gfCNCPoint4[28789] = {X 133.2007, Y 6.4835, Z -6.3333, A 0.000, B 0.000, C 0.000 }
gfCNCPoint4[28790] = {X 133.8833, Y 6.4837, Z -6.3333, A 0.000, B 0.000, C 0.000 }
gfCNCPoint4[28791] = {X 134.6792, Y 6.5720, Z -6.3333, A 0.000, B 0.000, C 0.000 }
gfCNCPoint4[28792] = {X 135.4415, Y 6.8171, Z -6.3333, A 0.000, B 0.000, C 0.000 }
gfCNCPoint4[28793] = {X 136.1397, Y 7.2091, Z -6.3333, A 0.000, B 0.000, C 0.000 }
gfCNCPoint4[28794] = {X 136.7458, Y 7.7322, Z -6.3333, A 0.000, B 0.000, C 0.000 }
gfCNCPoint4[28795] = {X 137.2357, Y 8.3657, Z -6.3333, A 0.000, B 0.000, C 0.000 }
gfCNCPoint4[28796] = {X 155.2276, Y 8.3657, Z -6.3333, A 0.000, B 0.000, C 0.000 }
gfCNCPoint4[28797] = {X 155.2814, Y 8.3748, Z -6.3333, A 0.000, B 0.000, C 0.000 }
gfCNCPoint4[28798] = {X 155.3395, Y 8.2839, Z -6.3333, A 0.000, B 0.000, C 0.000 }
gfCNCPoint4[28799] = {X 155.4001, Y 8.1946, Z -6.3333, A 0.000, B 0.000, C 0.000 }
gfCNCPoint4[28800] = {X 156.0394, Y 7.4794, Z -6.3333, A 0.000, B 0.000, C 0.000 }
gfCNCPoint4[28801] = {X 156.8306, Y 6.9370, Z -6.3333, A 0.000, B 0.000, C 0.000 }
gfCNCPoint4[28802] = {X 157.7282, Y 6.5985, Z -6.3333, A 0.000, B 0.000, C 0.000 }
gfCNCPoint4[28803] = {X 158.6805, Y 6.4835, Z -6.3333, A 0.000, B 0.000, C 0.000 }
gfCNCPoint4[28804] = {X 159.3739, Y 6.4839, Z -6.3333, A 0.000, B 0.000, C 0.000 }
gfCNCPoint4[28805] = {X 160.2554, Y 6.5939, Z -6.3333, A 0.000, B 0.000, C 0.000 }
gfCNCPoint4[28806] = {X 161.0909, Y 6.8959, Z -6.3333, A 0.000, B 0.000, C 0.000 }
gfCNCPoint4[28807] = {X 161.8391, Y 7.3747, Z -6.3333, A 0.000, B 0.000, C 0.000 }
gfCNCPoint4[28808] = {X 162.4632, Y 8.0070, Z -6.3333, A 0.000, B 0.000, C 0.000 }
gfCNCPoint4[28809] = {X 162.9324, Y 8.7613, Z -6.3333, A 0.000, B 0.000, C 0.000 }
gfCNCPoint4[28810] = {X 163.2234, Y 9.6007, Z -6.3333, A 0.000, B 0.000, C 0.000 }
gfCNCPoint4[28811] = {X 163.3221, Y 10.4835, Z -6.3333, A 0.000, B 0.000, C 0.000 }
gfCNCPoint4[28812] = {X 163.3221, Y 17.4615, Z -6.3333, A 0.000, B 0.000, C 0.000 }
gfCNCPoint4[28813] = {X 163.2218, Y 18.3516, Z -6.3333, A 0.000, B 0.000, C 0.000 }
gfCNCPoint4[28814] = {X 162.9260, Y 19.1971, Z -6.3333, A 0.000, B 0.000, C 0.000 }
gfCNCPoint4[28815] = {X 162.4494, Y 19.9555, Z -6.3333, A 0.000, B 0.000, C 0.000 }
gfCNCPoint4[28816] = {X 161.8160, Y 20.5889, Z -6.3333, A 0.000, B 0.000, C 0.000 }
gfCNCPoint4[28817] = {X 161.0576, Y 21.0654, Z -6.3333, A 0.000, B 0.000, C 0.000 }
gfCNCPoint4[28818] = {X 160.2122, Y 21.3613, Z -6.3333, A 0.000, B 0.000, C 0.000 }
gfCNCPoint4[28819] = {X 159.3221, Y 21.4615, Z -6.3333, A 0.000, B 0.000, C 0.000 }
gfCNCPoint4[28820] = {X 158.6805, Y 21.4615, Z -6.3333, A 0.000, B 0.000, C 0.000 }
gfCNCPoint4[28821] = {X 157.8710, Y 21.3764, Z -6.3333, A 0.000, B 0.000, C 0.000 }
gfCNCPoint4[28822] = {X 157.0951, Y 21.1304, Z -6.3333, A 0.000, B 0.000, C 0.000 }
gfCNCPoint4[28823] = {X 156.3845, Y 20.7335, Z -6.3333, A 0.000, B 0.000, C 0.000 }
gfCNCPoint4[28824] = {X 155.7680, Y 20.2020, Z -6.3333, A 0.000, B 0.000, C 0.000 }
gfCNCPoint4[28825] = {X 155.2709, Y 19.5575, Z -6.3333, A 0.000, B 0.000, C 0.000 }
gfCNCPoint4[28826] = {X 151.9570, Y 19.5587, Z -6.3333, A 0.000, B 0.000, C 0.000 }
gfCNCPoint4[28827] = {X 151.9558, Y 40.9999, Z -6.3333, A 0.000, B 0.000, C 0.000 }
gfCNCPoint4[28828] = {X 152.5009, Y 41.5868, Z -6.3333, A 0.000, B 0.000, C 0.000 }
gfCNCPoint4[28829] = {X 152.5894, Y 41.6922, Z -6.3333, A 0.000, B 0.000, C 0.000 }
gfCNCPoint4[28830] = {X 153.0754, Y 42.4562, Z -6.3333, A 0.000, B 0.000, C 0.000 }
gfCNCPoint4[28831] = {X 153.3784, Y 43.3095, Z -6.3333, A 0.000, B 0.000, C 0.000 }
gfCNCPoint4[28832] = {X 153.4831, Y 44.2089, Z -6.3333, A 0.000, B 0.000, C 0.000 }
gfCNCPoint4[28833] = {X 153.4829, Y 45.0384, Z -6.3333, A 0.000, B 0.000, C 0.000 }
gfCNCPoint4[28834] = {X 153.3753, Y 45.9222, Z -6.3333, A 0.000, B 0.000, C 0.000 }
gfCNCPoint4[28835] = {X 153.0750, Y 46.7602, Z -6.3333, A 0.000, B 0.000, C 0.000 }
gfCNCPoint4[28836] = {X 152.5967, Y 47.5111, Z -6.3333, A 0.000, B 0.000, C 0.000 }
gfCNCPoint4[28837] = {X 151.9642, Y 48.1376, Z -6.3333, A 0.000, B 0.000, C 0.000 }
gfCNCPoint4[28838] = {X 151.2087, Y 48.6086, Z -6.3333, A 0.000, B 0.000, C 0.000 }
gfCNCPoint4[28839] = {X 150.3678, Y 48.9009, Z -6.3333, A 0.000, B 0.000, C 0.000 }
gfCNCPoint4[28840] = {X 149.4831, Y 49.0000, Z -6.3333, A 0.000, B 0.000, C 0.000 }
gfCNCPoint4[28841] = {X 143.0396, Y 49.0000, Z -6.3333, A 0.000, B 0.000, C 0.000 }
gfCNCPoint4[28842] = {X 142.1495, Y 48.8997, Z -6.3333, A 0.000, B 0.000, C 0.000 }
gfCNCPoint4[28843] = {X 141.3041, Y 48.6039, Z -6.3333, A 0.000, B 0.000, C 0.000 }
gfCNCPoint4[28844] = {X 140.5457, Y 48.1273, Z -6.3333, A 0.000, B 0.000, C 0.000 }
gfCNCPoint4[28845] = {X 139.9123, Y 47.4939, Z -6.3333, A 0.000, B 0.000, C 0.000 }
gfCNCPoint4[28846] = {X 139.4357, Y 46.7355, Z -6.3333, A 0.000, B 0.000, C 0.000 }
gfCNCPoint4[28847] = {X 139.1399, Y 45.8901, Z -6.3333, A 0.000, B 0.000, C 0.000 }
gfCNCPoint4[28848] = {X 139.0396, Y 45.0000, Z -6.3333, A 0.000, B 0.000, C 0.000 }
gfCNCPoint4[28849] = {X 139.0400, Y 44.1538, Z -6.3333, A 0.000, B 0.000, C 0.000 }
gfCNCPoint4[28850] = {X 139.1506, Y 43.2730, Z -6.3333, A 0.000, B 0.000, C 0.000 }
gfCNCPoint4[28851] = {X 139.4528, Y 42.4382, Z -6.3333, A 0.000, B 0.000, C 0.000 }
gfCNCPoint4[28852] = {X 139.9317, Y 41.6907, Z -6.3333, A 0.000, B 0.000, C 0.000 }
gfCNCPoint4[28853] = {X 140.5636, Y 41.0672, Z -6.3333, A 0.000, B 0.000, C 0.000 }
gfCNCPoint4[28854] = {X 140.5636, Y 30.3968, Z -6.3333, A 0.000, B 0.000, C 0.000 }
gfCNCPoint4[28855] = {X 136.4836, Y 30.3968, Z -6.3333, A 0.000, B 0.000, C 0.000 }
gfCNCPoint4[28856] = {X 136.4836, Y 30.3968, Z -3.3333, A 0.000, B 0.000, C 0.000 }
gfCNCPoint4[28857] = {X 136.4836, Y 30.3968, Z 11.0000, A 0.000, B 0.000, C 0.000 }
gfCNCPoint4[28858] = {X 137.6634, Y 74.8921, Z 11.0000, A 0.000, B 0.000, C 0.000 }
gfCNCPoint4[28859] = {X 137.6634, Y 74.8921, Z -3.3333, A 0.000, B 0.000, C 0.000 }
gfCNCPoint4[28860] = {X 137.6634, Y 74.8921, Z -6.3333, A 0.000, B 0.000, C 0.000 }
gfCNCPoint4[28861] = {X 140.6800, Y 77.6392, Z -6.3333, A 0.000, B 0.000, C 0.000 }
gfCNCPoint4[28862] = {X 155.6321, Y 61.2197, Z -6.3333, A 0.000, B 0.000, C 0.000 }
gfCNCPoint4[28863] = {X 155.2773, Y 60.5141, Z -6.3333, A 0.000, B 0.000, C 0.000 }
gfCNCPoint4[28864] = {X 155.0568, Y 59.7556, Z -6.3333, A 0.000, B 0.000, C 0.000 }
gfCNCPoint4[28865] = {X 154.9781, Y 58.9697, Z -6.3333, A 0.000, B 0.000, C 0.000 }
gfCNCPoint4[28866] = {X 154.9780, Y 58.0000, Z -6.3333, A 0.000, B 0.000, C 0.000 }
gfCNCPoint4[28867] = {X 155.0863, Y 57.0387, Z -6.3333, A 0.000, B 0.000, C 0.000 }
gfCNCPoint4[28868] = {X 155.4058, Y 56.1256, Z -6.3333, A 0.000, B 0.000, C 0.000 }
gfCNCPoint4[28869] = {X 155.9204, Y 55.3065, Z -6.3333, A 0.000, B 0.000, C 0.000 }
gfCNCPoint4[28870] = {X 156.6045, Y 54.6225, Z -6.3333, A 0.000, B 0.000, C 0.000 }
gfCNCPoint4[28871] = {X 157.4236, Y 54.1078, Z -6.3333, A 0.000, B 0.000, C 0.000 }
gfCNCPoint4[28872] = {X 158.3367, Y 53.7883, Z -6.3333, A 0.000, B 0.000, C 0.000 }
gfCNCPoint4[28873] = {X 159.2980, Y 53.6800, Z -6.3333, A 0.000, B 0.000, C 0.000 }
gfCNCPoint4[28874] = {X 178.5335, Y 53.6800, Z -6.3333, A 0.000, B 0.000, C 0.000 }
gfCNCPoint4[28875] = {X 179.4948, Y 53.7883, Z -6.3333, A 0.000, B 0.000, C 0.000 }
gfCNCPoint4[28876] = {X 180.4079, Y 54.1078, Z -6.3333, A 0.000, B 0.000, C 0.000 }
gfCNCPoint4[28877] = {X 181.2270, Y 54.6225, Z -6.3333, A 0.000, B 0.000, C 0.000 }
gfCNCPoint4[28878] = {X 181.9110, Y 55.3065, Z -6.3333, A 0.000, B 0.000, C 0.000 }
gfCNCPoint4[28879] = {X 182.4257, Y 56.1256, Z -6.3333, A 0.000, B 0.000, C 0.000 }
gfCNCPoint4[28880] = {X 182.7452, Y 57.0387, Z -6.3333, A 0.000, B 0.000, C 0.000 }
gfCNCPoint4[28881] = {X 182.8535, Y 58.0000, Z -6.3333, A 0.000, B 0.000, C 0.000 }
gfCNCPoint4[28882] = {X 182.8535, Y 58.9342, Z -6.3333, A 0.000, B 0.000, C 0.000 }
gfCNCPoint4[28883] = {X 182.7808, Y 59.7231, Z -6.3333, A 0.000, B 0.000, C 0.000 }
gfCNCPoint4[28884] = {X 182.5653, Y 60.4855, Z -6.3333, A 0.000, B 0.000, C 0.000 }
gfCNCPoint4[28885] = {X 182.2142, Y 61.1956, Z -6.3333, A 0.000, B 0.000, C 0.000 }
gfCNCPoint4[28886] = {X 209.4796, Y 90.9543, Z -6.3333, A 0.000, B 0.000, C 0.000 }
gfCNCPoint4[28887] = {X 210.1361, Y 91.6204, Z -6.3333, A 0.000, B 0.000, C 0.000 }
gfCNCPoint4[28888] = {X 210.8392, Y 92.2369, Z -6.3333, A 0.000, B 0.000, C 0.000 }
gfCNCPoint4[28889] = {X 211.1136, Y 92.4105, Z -6.3333, A 0.000, B 0.000, C 0.000 }
gfCNCPoint4[28890] = {X 211.4212, Y 92.5146, Z -6.3333, A 0.000, B 0.000, C 0.000 }
gfCNCPoint4[28891] = {X 213.4040, Y 92.8239, Z -6.3333, A 0.000, B 0.000, C 0.000 }
gfCNCPoint4[28892] = {X 214.4546, Y 92.7351, Z -6.3333, A 0.000, B 0.000, C 0.000 }
gfCNCPoint4[28893] = {X 215.5073, Y 92.6749, Z -6.3333, A 0.000, B 0.000, C 0.000 }
gfCNCPoint4[28894] = {X 216.1774, Y 92.6018, Z -6.3333, A 0.000, B 0.000, C 0.000 }
gfCNCPoint4[28895] = {X 216.8226, Y 92.4068, Z -6.3333, A 0.000, B 0.000, C 0.000 }
gfCNCPoint4[28896] = {X 217.4209, Y 92.0964, Z -6.3333, A 0.000, B 0.000, C 0.000 }
gfCNCPoint4[28897] = {X 222.9613, Y 88.5209, Z -6.3333, A 0.000, B 0.000, C 0.000 }
gfCNCPoint4[28898] = {X 245.8274, Y 73.8996, Z -6.3333, A 0.000, B 0.000, C 0.000 }
gfCNCPoint4[28899] = {X 221.6306, Y 64.4044, Z -6.3333, A 0.000, B 0.000, C 0.000 }
gfCNCPoint4[28900] = {X 219.8631, Y 63.8129, Z -6.3333, A 0.000, B 0.000, C 0.000 }
gfCNCPoint4[28901] = {X 218.0397, Y 63.4269, Z -6.3333, A 0.000, B 0.000, C 0.000 }
gfCNCPoint4[28902] = {X 216.1841, Y 63.2516, Z -6.3333, A 0.000, B 0.000, C 0.000 }
gfCNCPoint4[28903] = {X 215.2523, Y 63.1173, Z -6.3333, A 0.000, B 0.000, C 0.000 }
gfCNCPoint4[28904] = {X 214.3716, Y 62.7843, Z -6.3333, A 0.000, B 0.000, C 0.000 }
gfCNCPoint4[28905] = {X 213.5841, Y 62.2684, Z -6.3333, A 0.000, B 0.000, C 0.000 }
gfCNCPoint4[28906] = {X 212.9270, Y 61.5942, Z -6.3333, A 0.000, B 0.000, C 0.000 }
gfCNCPoint4[28907] = {X 212.4315, Y 60.7936, Z -6.3333, A 0.000, B 0.000, C 0.000 }
gfCNCPoint4[28908] = {X 212.1213, Y 59.9047, Z -6.3333, A 0.000, B 0.000, C 0.000 }
gfCNCPoint4[28909] = {X 212.0110, Y 58.9697, Z -6.3333, A 0.000, B 0.000, C 0.000 }
gfCNCPoint4[28910] = {X 212.0108, Y 58.0000, Z -6.3333, A 0.000, B 0.000, C 0.000 }
gfCNCPoint4[28911] = {X 212.1191, Y 57.0387, Z -6.3333, A 0.000, B 0.000, C 0.000 }
gfCNCPoint4[28912] = {X 212.4386, Y 56.1256, Z -6.3333, A 0.000, B 0.000, C 0.000 }
gfCNCPoint4[28913] = {X 212.9533, Y 55.3065, Z -6.3333, A 0.000, B 0.000, C 0.000 }
gfCNCPoint4[28914] = {X 213.6373, Y 54.6225, Z -6.3333, A 0.000, B 0.000, C 0.000 }
gfCNCPoint4[28915] = {X 214.4564, Y 54.1078, Z -6.3333, A 0.000, B 0.000, C 0.000 }
gfCNCPoint4[28916] = {X 215.3695, Y 53.7883, Z -6.3333, A 0.000, B 0.000, C 0.000 }
gfCNCPoint4[28917] = {X 216.3308, Y 53.6800, Z -6.3333, A 0.000, B 0.000, C 0.000 }
gfCNCPoint4[28918] = {X 237.2617, Y 53.6800, Z -6.3333, A 0.000, B 0.000, C 0.000 }
gfCNCPoint4[28919] = {X 238.2230, Y 53.7883, Z -6.3333, A 0.000, B 0.000, C 0.000 }
gfCNCPoint4[28920] = {X 239.1361, Y 54.1078, Z -6.3333, A 0.000, B 0.000, C 0.000 }
gfCNCPoint4[28921] = {X 239.9552, Y 54.6225, Z -6.3333, A 0.000, B 0.000, C 0.000 }
gfCNCPoint4[28922] = {X 240.6392, Y 55.3065, Z -6.3333, A 0.000, B 0.000, C 0.000 }
gfCNCPoint4[28923] = {X 241.1539, Y 56.1256, Z -6.3333, A 0.000, B 0.000, C 0.000 }
gfCNCPoint4[28924] = {X 241.4734, Y 57.0387, Z -6.3333, A 0.000, B 0.000, C 0.000 }
gfCNCPoint4[28925] = {X 241.5817, Y 58.0000, Z -6.3333, A 0.000, B 0.000, C 0.000 }
gfCNCPoint4[28926] = {X 241.5817, Y 58.2319, Z -6.3333, A 0.000, B 0.000, C 0.000 }
gfCNCPoint4[28927] = {X 248.1145, Y 60.7793, Z -6.3333, A 0.000, B 0.000, C 0.000 }
gfCNCPoint4[28928] = {X 275.6322, Y 71.7016, Z -6.3333, A 0.000, B 0.000, C 0.000 }
gfCNCPoint4[28929] = {X 275.6336, Y 63.2123, Z -6.3333, A 0.000, B 0.000, C 0.000 }
gfCNCPoint4[28930] = {X 274.7820, Y 63.0032, Z -6.3333, A 0.000, B 0.000, C 0.000 }
gfCNCPoint4[28931] = {X 273.9901, Y 62.6264, Z -6.3333, A 0.000, B 0.000, C 0.000 }
gfCNCPoint4[28932] = {X 273.2907, Y 62.0974, Z -6.3333, A 0.000, B 0.000, C 0.000 }
gfCNCPoint4[28933] = {X 272.7125, Y 61.4381, Z -6.3333, A 0.000, B 0.000, C 0.000 }
gfCNCPoint4[28934] = {X 272.2793, Y 60.6756, Z -6.3333, A 0.000, B 0.000, C 0.000 }
gfCNCPoint4[28935] = {X 272.0090, Y 59.8414, Z -6.3333, A 0.000, B 0.000, C 0.000 }
gfCNCPoint4[28936] = {X 271.9128, Y 58.9697, Z -6.3333, A 0.000, B 0.000, C 0.000 }
gfCNCPoint4[28937] = {X 271.9127, Y 58.0000, Z -6.3333, A 0.000, B 0.000, C 0.000 }
gfCNCPoint4[28938] = {X 272.0210, Y 57.0387, Z -6.3333, A 0.000, B 0.000, C 0.000 }
gfCNCPoint4[28939] = {X 272.3405, Y 56.1256, Z -6.3333, A 0.000, B 0.000, C 0.000 }
gfCNCPoint4[28940] = {X 272.8552, Y 55.3065, Z -6.3333, A 0.000, B 0.000, C 0.000 }
gfCNCPoint4[28941] = {X 273.5392, Y 54.6225, Z -6.3333, A 0.000, B 0.000, C 0.000 }
gfCNCPoint4[28942] = {X 274.3583, Y 54.1078, Z -6.3333, A 0.000, B 0.000, C 0.000 }
gfCNCPoint4[28943] = {X 275.2714, Y 53.7883, Z -6.3333, A 0.000, B 0.000, C 0.000 }
gfCNCPoint4[28944] = {X 276.2327, Y 53.6800, Z -6.3333, A 0.000, B 0.000, C 0.000 }
gfCNCPoint4[28945] = {X 292.7731, Y 53.6800, Z -6.3333, A 0.000, B 0.000, C 0.000 }
gfCNCPoint4[28946] = {X 293.7344, Y 53.7883, Z -6.3333, A 0.000, B 0.000, C 0.000 }
gfCNCPoint4[28947] = {X 294.6475, Y 54.1078, Z -6.3333, A 0.000, B 0.000, C 0.000 }
gfCNCPoint4[28948] = {X 295.4666, Y 54.6225, Z -6.3333, A 0.000, B 0.000, C 0.000 }
gfCNCPoint4[28949] = {X 296.1506, Y 55.3065, Z -6.3333, A 0.000, B 0.000, C 0.000 }
gfCNCPoint4[28950] = {X 296.6653, Y 56.1256, Z -6.3333, A 0.000, B 0.000, C 0.000 }
gfCNCPoint4[28951] = {X 296.9848, Y 57.0387, Z -6.3333, A 0.000, B 0.000, C 0.000 }
gfCNCPoint4[28952] = {X 297.0931, Y 58.0000, Z -6.3333, A 0.000, B 0.000, C 0.000 }
gfCNCPoint4[28953] = {X 297.0931, Y 58.9350, Z -6.3333, A 0.000, B 0.000, C 0.000 }
gfCNCPoint4[28954] = {X 296.9713, Y 59.9431, Z -6.3333, A 0.000, B 0.000, C 0.000 }
gfCNCPoint4[28955] = {X 296.6183, Y 60.8953, Z -6.3333, A 0.000, B 0.000, C 0.000 }
gfCNCPoint4[28956] = {X 296.0536, Y 61.7393, Z -6.3333, A 0.000, B 0.000, C 0.000 }
gfCNCPoint4[28957] = {X 295.3082, Y 62.4288, Z -6.3333, A 0.000, B 0.000, C 0.000 }
gfCNCPoint4[28958] = {X 294.4227, Y 62.9260, Z -6.3333, A 0.000, B 0.000, C 0.000 }
gfCNCPoint4[28959] = {X 293.4460, Y 63.2036, Z -6.3333, A 0.000, B 0.000, C 0.000 }
gfCNCPoint4[28960] = {X 293.3735, Y 63.2251, Z -6.3333, A 0.000, B 0.000, C 0.000 }
gfCNCPoint4[28961] = {X 293.3847, Y 92.7805, Z -6.3333, A 0.000, B 0.000, C 0.000 }
gfCNCPoint4[28962] = {X 294.2373, Y 92.9980, Z -6.3333, A 0.000, B 0.000, C 0.000 }
gfCNCPoint4[28963] = {X 295.0288, Y 93.3825, Z -6.3333, A 0.000, B 0.000, C 0.000 }
gfCNCPoint4[28964] = {X 295.7267, Y 93.9184, Z -6.3333, A 0.000, B 0.000, C 0.000 }
gfCNCPoint4[28965] = {X 296.3026, Y 94.5837, Z -6.3333, A 0.000, B 0.000, C 0.000 }
gfCNCPoint4[28966] = {X 296.7329, Y 95.3512, Z -6.3333, A 0.000, B 0.000, C 0.000 }
gfCNCPoint4[28967] = {X 297.0000, Y 96.1896, Z -6.3333, A 0.000, B 0.000, C 0.000 }
gfCNCPoint4[28968] = {X 297.0931, Y 97.0645, Z -6.3333, A 0.000, B 0.000, C 0.000 }
gfCNCPoint4[28969] = {X 297.0931, Y 98.0000, Z -6.3333, A 0.000, B 0.000, C 0.000 }
gfCNCPoint4[28970] = {X 296.9848, Y 98.9613, Z -6.3333, A 0.000, B 0.000, C 0.000 }
gfCNCPoint4[28971] = {X 296.6653, Y 99.8744, Z -6.3333, A 0.000, B 0.000, C 0.000 }
gfCNCPoint4[28972] = {X 296.1506, Y 100.6935, Z -6.3333, A 0.000, B 0.000, C 0.000 }
gfCNCPoint4[28973] = {X 295.4666, Y 101.3775, Z -6.3333, A 0.000, B 0.000, C 0.000 }
gfCNCPoint4[28974] = {X 294.6475, Y 101.8922, Z -6.3333, A 0.000, B 0.000, C 0.000 }
gfCNCPoint4[28975] = {X 293.7344, Y 102.2117, Z -6.3333, A 0.000, B 0.000, C 0.000 }
gfCNCPoint4[28976] = {X 292.7731, Y 102.3200, Z -6.3333, A 0.000, B 0.000, C 0.000 }
gfCNCPoint4[28977] = {X 276.2327, Y 102.3200, Z -6.3333, A 0.000, B 0.000, C 0.000 }
gfCNCPoint4[28978] = {X 275.2714, Y 102.2117, Z -6.3333, A 0.000, B 0.000, C 0.000 }
gfCNCPoint4[28979] = {X 274.3583, Y 101.8922, Z -6.3333, A 0.000, B 0.000, C 0.000 }
gfCNCPoint4[28980] = {X 273.5392, Y 101.3775, Z -6.3333, A 0.000, B 0.000, C 0.000 }
gfCNCPoint4[28981] = {X 272.8552, Y 100.6935, Z -6.3333, A 0.000, B 0.000, C 0.000 }
gfCNCPoint4[28982] = {X 272.3405, Y 99.8744, Z -6.3333, A 0.000, B 0.000, C 0.000 }
gfCNCPoint4[28983] = {X 272.0210, Y 98.9613, Z -6.3333, A 0.000, B 0.000, C 0.000 }
gfCNCPoint4[28984] = {X 271.9127, Y 98.0000, Z -6.3333, A 0.000, B 0.000, C 0.000 }
gfCNCPoint4[28985] = {X 271.9127, Y 97.0659, Z -6.3333, A 0.000, B 0.000, C 0.000 }
gfCNCPoint4[28986] = {X 272.0026, Y 96.1891, Z -6.3333, A 0.000, B 0.000, C 0.000 }
gfCNCPoint4[28987] = {X 272.2686, Y 95.3488, Z -6.3333, A 0.000, B 0.000, C 0.000 }
gfCNCPoint4[28988] = {X 272.6997, Y 94.5800, Z -6.3333, A 0.000, B 0.000, C 0.000 }
gfCNCPoint4[28989] = {X 273.2777, Y 93.9146, Z -6.3333, A 0.000, B 0.000, C 0.000 }
gfCNCPoint4[28990] = {X 273.9788, Y 93.3805, Z -6.3333, A 0.000, B 0.000, C 0.000 }
gfCNCPoint4[28991] = {X 274.7737, Y 92.9997, Z -6.3333, A 0.000, B 0.000, C 0.000 }
gfCNCPoint4[28992] = {X 275.6294, Y 92.7883, Z -6.3333, A 0.000, B 0.000, C 0.000 }
gfCNCPoint4[28993] = {X 275.6294, Y 85.5950, Z -6.3333, A 0.000, B 0.000, C 0.000 }
gfCNCPoint4[28994] = {X 262.6398, Y 80.5030, Z -6.3333, A 0.000, B 0.000, C 0.000 }
gfCNCPoint4[28995] = {X 262.2779, Y 80.7315, Z -6.3333, A 0.000, B 0.000, C 0.000 }
gfCNCPoint4[28996] = {X 237.7972, Y 96.5883, Z -6.3333, A 0.000, B 0.000, C 0.000 }
gfCNCPoint4[28997] = {X 237.7998, Y 97.0650, Z -6.3333, A 0.000, B 0.000, C 0.000 }
gfCNCPoint4[28998] = {X 237.7998, Y 98.0000, Z -6.3333, A 0.000, B 0.000, C 0.000 }
gfCNCPoint4[28999] = {X 237.6915, Y 98.9613, Z -6.3333, A 0.000, B 0.000, C 0.000 }
gfCNCPoint4[29000] = {X 237.3720, Y 99.8744, Z -6.3333, A 0.000, B 0.000, C 0.000 }
gfCNCPoint4[29001] = {X 236.8573, Y 100.6935, Z -6.3333, A 0.000, B 0.000, C 0.000 }
gfCNCPoint4[29002] = {X 236.1733, Y 101.3775, Z -6.3333, A 0.000, B 0.000, C 0.000 }
gfCNCPoint4[29003] = {X 235.3542, Y 101.8922, Z -6.3333, A 0.000, B 0.000, C 0.000 }
gfCNCPoint4[29004] = {X 234.4411, Y 102.2117, Z -6.3333, A 0.000, B 0.000, C 0.000 }
gfCNCPoint4[29005] = {X 233.4798, Y 102.3200, Z -6.3333, A 0.000, B 0.000, C 0.000 }
gfCNCPoint4[29006] = {X 214.1790, Y 102.3200, Z -6.3333, A 0.000, B 0.000, C 0.000 }
gfCNCPoint4[29007] = {X 213.7862, Y 102.3021, Z -6.3333, A 0.000, B 0.000, C 0.000 }
gfCNCPoint4[29008] = {X 213.3966, Y 102.2485, Z -6.3333, A 0.000, B 0.000, C 0.000 }
gfCNCPoint4[29009] = {X 213.0070, Y 102.3021, Z -6.3333, A 0.000, B 0.000, C 0.000 }
gfCNCPoint4[29010] = {X 212.6141, Y 102.3200, Z -6.3333, A 0.000, B 0.000, C 0.000 }
gfCNCPoint4[29011] = {X 194.9870, Y 102.3200, Z -6.3333, A 0.000, B 0.000, C 0.000 }
gfCNCPoint4[29012] = {X 194.0257, Y 102.2117, Z -6.3333, A 0.000, B 0.000, C 0.000 }
gfCNCPoint4[29013] = {X 193.1126, Y 101.8922, Z -6.3333, A 0.000, B 0.000, C 0.000 }
gfCNCPoint4[29014] = {X 192.2935, Y 101.3775, Z -6.3333, A 0.000, B 0.000, C 0.000 }
gfCNCPoint4[29015] = {X 191.6094, Y 100.6935, Z -6.3333, A 0.000, B 0.000, C 0.000 }
gfCNCPoint4[29016] = {X 191.0948, Y 99.8744, Z -6.3333, A 0.000, B 0.000, C 0.000 }
gfCNCPoint4[29017] = {X 190.7753, Y 98.9613, Z -6.3333, A 0.000, B 0.000, C 0.000 }
gfCNCPoint4[29018] = {X 190.6670, Y 98.0000, Z -6.3333, A 0.000, B 0.000, C 0.000 }
gfCNCPoint4[29019] = {X 190.6670, Y 97.0659, Z -6.3333, A 0.000, B 0.000, C 0.000 }
gfCNCPoint4[29020] = {X 190.7727, Y 96.1162, Z -6.3333, A 0.000, B 0.000, C 0.000 }
gfCNCPoint4[29021] = {X 191.0846, Y 95.2129, Z -6.3333, A 0.000, B 0.000, C 0.000 }
gfCNCPoint4[29022] = {X 191.5874, Y 94.4003, Z -6.3333, A 0.000, B 0.000, C 0.000 }
gfCNCPoint4[29023] = {X 188.5647, Y 91.1002, Z -6.3333, A 0.000, B 0.000, C 0.000 }
gfCNCPoint4[29024] = {X 150.0898, Y 91.1002, Z -6.3333, A 0.000, B 0.000, C 0.000 }
gfCNCPoint4[29025] = {X 147.1454, Y 94.3623, Z -6.3333, A 0.000, B 0.000, C 0.000 }
gfCNCPoint4[29026] = {X 147.6646, Y 95.1836, Z -6.3333, A 0.000, B 0.000, C 0.000 }
gfCNCPoint4[29027] = {X 147.9879, Y 96.1000, Z -6.3333, A 0.000, B 0.000, C 0.000 }
gfCNCPoint4[29028] = {X 148.0991, Y 97.0653, Z -6.3333, A 0.000, B 0.000, C 0.000 }
gfCNCPoint4[29029] = {X 148.0991, Y 98.0000, Z -6.3333, A 0.000, B 0.000, C 0.000 }
gfCNCPoint4[29030] = {X 147.9908, Y 98.9613, Z -6.3333, A 0.000, B 0.000, C 0.000 }
gfCNCPoint4[29031] = {X 147.6713, Y 99.8744, Z -6.3333, A 0.000, B 0.000, C 0.000 }
gfCNCPoint4[29032] = {X 147.1566, Y 100.6935, Z -6.3333, A 0.000, B 0.000, C 0.000 }
gfCNCPoint4[29033] = {X 146.4726, Y 101.3775, Z -6.3333, A 0.000, B 0.000, C 0.000 }
gfCNCPoint4[29034] = {X 145.6535, Y 101.8922, Z -6.3333, A 0.000, B 0.000, C 0.000 }
gfCNCPoint4[29035] = {X 144.7404, Y 102.2117, Z -6.3333, A 0.000, B 0.000, C 0.000 }
gfCNCPoint4[29036] = {X 143.7791, Y 102.3200, Z -6.3333, A 0.000, B 0.000, C 0.000 }
gfCNCPoint4[29037] = {X 125.0000, Y 102.3200, Z -6.3333, A 0.000, B 0.000, C 0.000 }
gfCNCPoint4[29038] = {X 124.0387, Y 102.2117, Z -6.3333, A 0.000, B 0.000, C 0.000 }
gfCNCPoint4[29039] = {X 123.1256, Y 101.8922, Z -6.3333, A 0.000, B 0.000, C 0.000 }
gfCNCPoint4[29040] = {X 122.3065, Y 101.3775, Z -6.3333, A 0.000, B 0.000, C 0.000 }
gfCNCPoint4[29041] = {X 121.6225, Y 100.6935, Z -6.3333, A 0.000, B 0.000, C 0.000 }
gfCNCPoint4[29042] = {X 121.1078, Y 99.8744, Z -6.3333, A 0.000, B 0.000, C 0.000 }
gfCNCPoint4[29043] = {X 120.7883, Y 98.9613, Z -6.3333, A 0.000, B 0.000, C 0.000 }
gfCNCPoint4[29044] = {X 120.6800, Y 98.0000, Z -6.3333, A 0.000, B 0.000, C 0.000 }
gfCNCPoint4[29045] = {X 120.6800, Y 97.0659, Z -6.3333, A 0.000, B 0.000, C 0.000 }
gfCNCPoint4[29046] = {X 120.7832, Y 96.1275, Z -6.3333, A 0.000, B 0.000, C 0.000 }
gfCNCPoint4[29047] = {X 121.0877, Y 95.2340, Z -6.3333, A 0.000, B 0.000, C 0.000 }
gfCNCPoint4[29048] = {X 121.5790, Y 94.4279, Z -6.3333, A 0.000, B 0.000, C 0.000 }
gfCNCPoint4[29049] = {X 122.2338, Y 93.7478, Z -6.3333, A 0.000, B 0.000, C 0.000 }
gfCNCPoint4[29050] = {X 123.0206, Y 93.2261, Z -6.3333, A 0.000, B 0.000, C 0.000 }
gfCNCPoint4[29051] = {X 123.9019, Y 92.8878, Z -6.3333, A 0.000, B 0.000, C 0.000 }
gfCNCPoint4[29052] = {X 124.8357, Y 92.7491, Z -6.3333, A 0.000, B 0.000, C 0.000 }
gfCNCPoint4[29053] = {X 124.8807, Y 92.7315, Z -6.3333, A 0.000, B 0.000, C 0.000 }
gfCNCPoint4[29054] = {X 124.9278, Y 92.7208, Z -6.3333, A 0.000, B 0.000, C 0.000 }
gfCNCPoint4[29055] = {X 125.4494, Y 92.6434, Z -6.3333, A 0.000, B 0.000, C 0.000 }
gfCNCPoint4[29056] = {X 126.2804, Y 92.5036, Z -6.3333, A 0.000, B 0.000, C 0.000 }
gfCNCPoint4[29057] = {X 127.0999, Y 92.3072, Z -6.3333, A 0.000, B 0.000, C 0.000 }
gfCNCPoint4[29058] = {X 128.3213, Y 91.1562, Z -6.3333, A 0.000, B 0.000, C 0.000 }
gfCNCPoint4[29059] = {X 129.4782, Y 89.9403, Z -6.3333, A 0.000, B 0.000, C 0.000 }
gfCNCPoint4[29060] = {X 140.6800, Y 77.6392, Z -6.3333, A 0.000, B 0.000, C 0.000 }
gfCNCPoint4[29061] = {X 137.7225, Y 74.9460, Z -6.3333, A 0.000, B 0.000, C 0.000 }
gfCNCPoint4[29062] = {X 140.7391, Y 77.6930, Z -6.3333, A 0.000, B 0.000, C 0.000 }
gfCNCPoint4[29063] = {X 155.7324, Y 61.2284, Z -6.3333, A 0.000, B 0.000, C 0.000 }
gfCNCPoint4[29064] = {X 155.3666, Y 60.5223, Z -6.3333, A 0.000, B 0.000, C 0.000 }
gfCNCPoint4[29065] = {X 155.1392, Y 59.7602, Z -6.3333, A 0.000, B 0.000, C 0.000 }
gfCNCPoint4[29066] = {X 155.0581, Y 58.9691, Z -6.3333, A 0.000, B 0.000, C 0.000 }
gfCNCPoint4[29067] = {X 155.0580, Y 58.0000, Z -6.3333, A 0.000, B 0.000, C 0.000 }
gfCNCPoint4[29068] = {X 155.1643, Y 57.0565, Z -6.3333, A 0.000, B 0.000, C 0.000 }
gfCNCPoint4[29069] = {X 155.4778, Y 56.1603, Z -6.3333, A 0.000, B 0.000, C 0.000 }
gfCNCPoint4[29070] = {X 155.9830, Y 55.3564, Z -6.3333, A 0.000, B 0.000, C 0.000 }
gfCNCPoint4[29071] = {X 156.6544, Y 54.6850, Z -6.3333, A 0.000, B 0.000, C 0.000 }
gfCNCPoint4[29072] = {X 157.4583, Y 54.1799, Z -6.3333, A 0.000, B 0.000, C 0.000 }
gfCNCPoint4[29073] = {X 158.3545, Y 53.8663, Z -6.3333, A 0.000, B 0.000, C 0.000 }
gfCNCPoint4[29074] = {X 159.2980, Y 53.7600, Z -6.3333, A 0.000, B 0.000, C 0.000 }
gfCNCPoint4[29075] = {X 178.5335, Y 53.7600, Z -6.3333, A 0.000, B 0.000, C 0.000 }
gfCNCPoint4[29076] = {X 179.4770, Y 53.8663, Z -6.3333, A 0.000, B 0.000, C 0.000 }
gfCNCPoint4[29077] = {X 180.3732, Y 54.1799, Z -6.3333, A 0.000, B 0.000, C 0.000 }
gfCNCPoint4[29078] = {X 181.1771, Y 54.6850, Z -6.3333, A 0.000, B 0.000, C 0.000 }
gfCNCPoint4[29079] = {X 181.8485, Y 55.3564, Z -6.3333, A 0.000, B 0.000, C 0.000 }
gfCNCPoint4[29080] = {X 182.3536, Y 56.1603, Z -6.3333, A 0.000, B 0.000, C 0.000 }
gfCNCPoint4[29081] = {X 182.6672, Y 57.0565, Z -6.3333, A 0.000, B 0.000, C 0.000 }
gfCNCPoint4[29082] = {X 182.7735, Y 58.0000, Z -6.3333, A 0.000, B 0.000, C 0.000 }
gfCNCPoint4[29083] = {X 182.7735, Y 58.9342, Z -6.3333, A 0.000, B 0.000, C 0.000 }
gfCNCPoint4[29084] = {X 182.6985, Y 59.7282, Z -6.3333, A 0.000, B 0.000, C 0.000 }
gfCNCPoint4[29085] = {X 182.4761, Y 60.4941, Z -6.3333, A 0.000, B 0.000, C 0.000 }
gfCNCPoint4[29086] = {X 182.1142, Y 61.2048, Z -6.3333, A 0.000, B 0.000, C 0.000 }
gfCNCPoint4[29087] = {X 209.4206, Y 91.0084, Z -6.3333, A 0.000, B 0.000, C 0.000 }
gfCNCPoint4[29088] = {X 210.0812, Y 91.6786, Z -6.3333, A 0.000, B 0.000, C 0.000 }
gfCNCPoint4[29089] = {X 210.7887, Y 92.2989, Z -6.3333, A 0.000, B 0.000, C 0.000 }
gfCNCPoint4[29090] = {X 211.0801, Y 92.4832, Z -6.3333, A 0.000, B 0.000, C 0.000 }
gfCNCPoint4[29091] = {X 211.4068, Y 92.5933, Z -6.3333, A 0.000, B 0.000, C 0.000 }
gfCNCPoint4[29092] = {X 213.4017, Y 92.9045, Z -6.3333, A 0.000, B 0.000, C 0.000 }
gfCNCPoint4[29093] = {X 214.4547, Y 92.8153, Z -6.3333, A 0.000, B 0.000, C 0.000 }
gfCNCPoint4[29094] = {X 215.5097, Y 92.7549, Z -6.3333, A 0.000, B 0.000, C 0.000 }
gfCNCPoint4[29095] = {X 216.1941, Y 92.6801, Z -6.3333, A 0.000, B 0.000, C 0.000 }
gfCNCPoint4[29096] = {X 216.8531, Y 92.4807, Z -6.3333, A 0.000, B 0.000, C 0.000 }
gfCNCPoint4[29097] = {X 217.4643, Y 92.1637, Z -6.3333, A 0.000, B 0.000, C 0.000 }
gfCNCPoint4[29098] = {X 223.0046, Y 88.5882, Z -6.3333, A 0.000, B 0.000, C 0.000 }
gfCNCPoint4[29099] = {X 246.0027, Y 73.8825, Z -6.3333, A 0.000, B 0.000, C 0.000 }
gfCNCPoint4[29100] = {X 221.6603, Y 64.3301, Z -6.3333, A 0.000, B 0.000, C 0.000 }
gfCNCPoint4[29101] = {X 219.8841, Y 63.7357, Z -6.3333, A 0.000, B 0.000, C 0.000 }
gfCNCPoint4[29102] = {X 218.0517, Y 63.3478, Z -6.3333, A 0.000, B 0.000, C 0.000 }
gfCNCPoint4[29103] = {X 216.1870, Y 63.1716, Z -6.3333, A 0.000, B 0.000, C 0.000 }
gfCNCPoint4[29104] = {X 215.2724, Y 63.0398, Z -6.3333, A 0.000, B 0.000, C 0.000 }
gfCNCPoint4[29105] = {X 214.4080, Y 62.7130, Z -6.3333, A 0.000, B 0.000, C 0.000 }
gfCNCPoint4[29106] = {X 213.6350, Y 62.2067, Z -6.3333, A 0.000, B 0.000, C 0.000 }
gfCNCPoint4[29107] = {X 212.9900, Y 61.5450, Z -6.3333, A 0.000, B 0.000, C 0.000 }
gfCNCPoint4[29108] = {X 212.5038, Y 60.7592, Z -6.3333, A 0.000, B 0.000, C 0.000 }
gfCNCPoint4[29109] = {X 212.1992, Y 59.8868, Z -6.3333, A 0.000, B 0.000, C 0.000 }
gfCNCPoint4[29110] = {X 212.0910, Y 58.9691, Z -6.3333, A 0.000, B 0.000, C 0.000 }
gfCNCPoint4[29111] = {X 212.0908, Y 58.0000, Z -6.3333, A 0.000, B 0.000, C 0.000 }
gfCNCPoint4[29112] = {X 212.1971, Y 57.0565, Z -6.3333, A 0.000, B 0.000, C 0.000 }
gfCNCPoint4[29113] = {X 212.5107, Y 56.1603, Z -6.3333, A 0.000, B 0.000, C 0.000 }
gfCNCPoint4[29114] = {X 213.0158, Y 55.3564, Z -6.3333, A 0.000, B 0.000, C 0.000 }
gfCNCPoint4[29115] = {X 213.6872, Y 54.6850, Z -6.3333, A 0.000, B 0.000, C 0.000 }
gfCNCPoint4[29116] = {X 214.4911, Y 54.1799, Z -6.3333, A 0.000, B 0.000, C 0.000 }
gfCNCPoint4[29117] = {X 215.3873, Y 53.8663, Z -6.3333, A 0.000, B 0.000, C 0.000 }
gfCNCPoint4[29118] = {X 216.3308, Y 53.7600, Z -6.3333, A 0.000, B 0.000, C 0.000 }
gfCNCPoint4[29119] = {X 237.2617, Y 53.7600, Z -6.3333, A 0.000, B 0.000, C 0.000 }
gfCNCPoint4[29120] = {X 238.2052, Y 53.8663, Z -6.3333, A 0.000, B 0.000, C 0.000 }
gfCNCPoint4[29121] = {X 239.1014, Y 54.1799, Z -6.3333, A 0.000, B 0.000, C 0.000 }
gfCNCPoint4[29122] = {X 239.9053, Y 54.6850, Z -6.3333, A 0.000, B 0.000, C 0.000 }
gfCNCPoint4[29123] = {X 240.5767, Y 55.3564, Z -6.3333, A 0.000, B 0.000, C 0.000 }
gfCNCPoint4[29124] = {X 241.0818, Y 56.1603, Z -6.3333, A 0.000, B 0.000, C 0.000 }
gfCNCPoint4[29125] = {X 241.3954, Y 57.0565, Z -6.3333, A 0.000, B 0.000, C 0.000 }
gfCNCPoint4[29126] = {X 241.5017, Y 58.0000, Z -6.3333, A 0.000, B 0.000, C 0.000 }
gfCNCPoint4[29127] = {X 241.5017, Y 58.2866, Z -6.3333, A 0.000, B 0.000, C 0.000 }
gfCNCPoint4[29128] = {X 248.0852, Y 60.8537, Z -6.3333, A 0.000, B 0.000, C 0.000 }
gfCNCPoint4[29129] = {X 275.7122, Y 71.8194, Z -6.3333, A 0.000, B 0.000, C 0.000 }
gfCNCPoint4[29130] = {X 275.7136, Y 63.1422, Z -6.3333, A 0.000, B 0.000, C 0.000 }
gfCNCPoint4[29131] = {X 274.8651, Y 62.9475, Z -6.3333, A 0.000, B 0.000, C 0.000 }
gfCNCPoint4[29132] = {X 274.0742, Y 62.5835, Z -6.3333, A 0.000, B 0.000, C 0.000 }
gfCNCPoint4[29133] = {X 273.3744, Y 62.0658, Z -6.3333, A 0.000, B 0.000, C 0.000 }
gfCNCPoint4[29134] = {X 272.7950, Y 61.4160, Z -6.3333, A 0.000, B 0.000, C 0.000 }
gfCNCPoint4[29135] = {X 272.3606, Y 60.6616, Z -6.3333, A 0.000, B 0.000, C 0.000 }
gfCNCPoint4[29136] = {X 272.0894, Y 59.8343, Z -6.3333, A 0.000, B 0.000, C 0.000 }
gfCNCPoint4[29137] = {X 271.9928, Y 58.9691, Z -6.3333, A 0.000, B 0.000, C 0.000 }
gfCNCPoint4[29138] = {X 271.9927, Y 58.0000, Z -6.3333, A 0.000, B 0.000, C 0.000 }
gfCNCPoint4[29139] = {X 272.0990, Y 57.0565, Z -6.3333, A 0.000, B 0.000, C 0.000 }
gfCNCPoint4[29140] = {X 272.4126, Y 56.1603, Z -6.3333, A 0.000, B 0.000, C 0.000 }
gfCNCPoint4[29141] = {X 272.9177, Y 55.3564, Z -6.3333, A 0.000, B 0.000, C 0.000 }
gfCNCPoint4[29142] = {X 273.5891, Y 54.6850, Z -6.3333, A 0.000, B 0.000, C 0.000 }
gfCNCPoint4[29143] = {X 274.3930, Y 54.1799, Z -6.3333, A 0.000, B 0.000, C 0.000 }
gfCNCPoint4[29144] = {X 275.2892, Y 53.8663, Z -6.3333, A 0.000, B 0.000, C 0.000 }
gfCNCPoint4[29145] = {X 276.2327, Y 53.7600, Z -6.3333, A 0.000, B 0.000, C 0.000 }
gfCNCPoint4[29146] = {X 292.7731, Y 53.7600, Z -6.3333, A 0.000, B 0.000, C 0.000 }
gfCNCPoint4[29147] = {X 293.7166, Y 53.8663, Z -6.3333, A 0.000, B 0.000, C 0.000 }
gfCNCPoint4[29148] = {X 294.6128, Y 54.1799, Z -6.3333, A 0.000, B 0.000, C 0.000 }
gfCNCPoint4[29149] = {X 295.4167, Y 54.6850, Z -6.3333, A 0.000, B 0.000, C 0.000 }
gfCNCPoint4[29150] = {X 296.0881, Y 55.3564, Z -6.3333, A 0.000, B 0.000, C 0.000 }
gfCNCPoint4[29151] = {X 296.5932, Y 56.1603, Z -6.3333, A 0.000, B 0.000, C 0.000 }
gfCNCPoint4[29152] = {X 296.9068, Y 57.0565, Z -6.3333, A 0.000, B 0.000, C 0.000 }
gfCNCPoint4[29153] = {X 297.0131, Y 58.0000, Z -6.3333, A 0.000, B 0.000, C 0.000 }
gfCNCPoint4[29154] = {X 297.0131, Y 58.9348, Z -6.3333, A 0.000, B 0.000, C 0.000 }
gfCNCPoint4[29155] = {X 296.8933, Y 59.9252, Z -6.3333, A 0.000, B 0.000, C 0.000 }
gfCNCPoint4[29156] = {X 296.5463, Y 60.8604, Z -6.3333, A 0.000, B 0.000, C 0.000 }
gfCNCPoint4[29157] = {X 295.9912, Y 61.6893, Z -6.3333, A 0.000, B 0.000, C 0.000 }
gfCNCPoint4[29158] = {X 295.2583, Y 62.3661, Z -6.3333, A 0.000, B 0.000, C 0.000 }
gfCNCPoint4[29159] = {X 294.3881, Y 62.8538, Z -6.3333, A 0.000, B 0.000, C 0.000 }
gfCNCPoint4[29160] = {X 293.4282, Y 63.1255, Z -6.3333, A 0.000, B 0.000, C 0.000 }
gfCNCPoint4[29161] = {X 293.2934, Y 63.1654, Z -6.3333, A 0.000, B 0.000, C 0.000 }
gfCNCPoint4[29162] = {X 293.3048, Y 92.8500, Z -6.3333, A 0.000, B 0.000, C 0.000 }
gfCNCPoint4[29163] = {X 294.1543, Y 93.0532, Z -6.3333, A 0.000, B 0.000, C 0.000 }
gfCNCPoint4[29164] = {X 294.9447, Y 93.4250, Z -6.3333, A 0.000, B 0.000, C 0.000 }
gfCNCPoint4[29165] = {X 295.6431, Y 93.9498, Z -6.3333, A 0.000, B 0.000, C 0.000 }
gfCNCPoint4[29166] = {X 296.2201, Y 94.6056, Z -6.3333, A 0.000, B 0.000, C 0.000 }
gfCNCPoint4[29167] = {X 296.6516, Y 95.3650, Z -6.3333, A 0.000, B 0.000, C 0.000 }
gfCNCPoint4[29168] = {X 296.9197, Y 96.1964, Z -6.3333, A 0.000, B 0.000, C 0.000 }
gfCNCPoint4[29169] = {X 297.0131, Y 97.0649, Z -6.3333, A 0.000, B 0.000, C 0.000 }
gfCNCPoint4[29170] = {X 297.0131, Y 98.0000, Z -6.3333, A 0.000, B 0.000, C 0.000 }
gfCNCPoint4[29171] = {X 296.9068, Y 98.9435, Z -6.3333, A 0.000, B 0.000, C 0.000 }
gfCNCPoint4[29172] = {X 296.5932, Y 99.8397, Z -6.3333, A 0.000, B 0.000, C 0.000 }
gfCNCPoint4[29173] = {X 296.0881, Y 100.6436, Z -6.3333, A 0.000, B 0.000, C 0.000 }
gfCNCPoint4[29174] = {X 295.4167, Y 101.3150, Z -6.3333, A 0.000, B 0.000, C 0.000 }
gfCNCPoint4[29175] = {X 294.6128, Y 101.8201, Z -6.3333, A 0.000, B 0.000, C 0.000 }
gfCNCPoint4[29176] = {X 293.7166, Y 102.1337, Z -6.3333, A 0.000, B 0.000, C 0.000 }
gfCNCPoint4[29177] = {X 292.7731, Y 102.2400, Z -6.3333, A 0.000, B 0.000, C 0.000 }
gfCNCPoint4[29178] = {X 276.2327, Y 102.2400, Z -6.3333, A 0.000, B 0.000, C 0.000 }
gfCNCPoint4[29179] = {X 275.2892, Y 102.1337, Z -6.3333, A 0.000, B 0.000, C 0.000 }
gfCNCPoint4[29180] = {X 274.3930, Y 101.8201, Z -6.3333, A 0.000, B 0.000, C 0.000 }
gfCNCPoint4[29181] = {X 273.5891, Y 101.3150, Z -6.3333, A 0.000, B 0.000, C 0.000 }
gfCNCPoint4[29182] = {X 272.9177, Y 100.6436, Z -6.3333, A 0.000, B 0.000, C 0.000 }
gfCNCPoint4[29183] = {X 272.4126, Y 99.8397, Z -6.3333, A 0.000, B 0.000, C 0.000 }
gfCNCPoint4[29184] = {X 272.0990, Y 98.9435, Z -6.3333, A 0.000, B 0.000, C 0.000 }
gfCNCPoint4[29185] = {X 271.9927, Y 98.0000, Z -6.3333, A 0.000, B 0.000, C 0.000 }
gfCNCPoint4[29186] = {X 271.9927, Y 97.0659, Z -6.3333, A 0.000, B 0.000, C 0.000 }
gfCNCPoint4[29187] = {X 272.0830, Y 96.1956, Z -6.3333, A 0.000, B 0.000, C 0.000 }
gfCNCPoint4[29188] = {X 272.3500, Y 95.3624, Z -6.3333, A 0.000, B 0.000, C 0.000 }
gfCNCPoint4[29189] = {X 272.7823, Y 94.6017, Z -6.3333, A 0.000, B 0.000, C 0.000 }
gfCNCPoint4[29190] = {X 273.3615, Y 93.9460, Z -6.3333, A 0.000, B 0.000, C 0.000 }
gfCNCPoint4[29191] = {X 274.0630, Y 93.4231, Z -6.3333, A 0.000, B 0.000, C 0.000 }
gfCNCPoint4[29192] = {X 274.8569, Y 93.0553, Z -6.3333, A 0.000, B 0.000, C 0.000 }
gfCNCPoint4[29193] = {X 275.7094, Y 92.8584, Z -6.3333, A 0.000, B 0.000, C 0.000 }
gfCNCPoint4[29194] = {X 275.7094, Y 85.5404, Z -6.3333, A 0.000, B 0.000, C 0.000 }
gfCNCPoint4[29195] = {X 262.6313, Y 80.4138, Z -6.3333, A 0.000, B 0.000, C 0.000 }
gfCNCPoint4[29196] = {X 262.2347, Y 80.6641, Z -6.3333, A 0.000, B 0.000, C 0.000 }
gfCNCPoint4[29197] = {X 237.7169, Y 96.5449, Z -6.3333, A 0.000, B 0.000, C 0.000 }
gfCNCPoint4[29198] = {X 237.7198, Y 97.0652, Z -6.3333, A 0.000, B 0.000, C 0.000 }
gfCNCPoint4[29199] = {X 237.7198, Y 98.0000, Z -6.3333, A 0.000, B 0.000, C 0.000 }
gfCNCPoint4[29200] = {X 237.6135, Y 98.9435, Z -6.3333, A 0.000, B 0.000, C 0.000 }
gfCNCPoint4[29201] = {X 237.2999, Y 99.8397, Z -6.3333, A 0.000, B 0.000, C 0.000 }
gfCNCPoint4[29202] = {X 236.7948, Y 100.6436, Z -6.3333, A 0.000, B 0.000, C 0.000 }
gfCNCPoint4[29203] = {X 236.1234, Y 101.3150, Z -6.3333, A 0.000, B 0.000, C 0.000 }
gfCNCPoint4[29204] = {X 235.3195, Y 101.8201, Z -6.3333, A 0.000, B 0.000, C 0.000 }
gfCNCPoint4[29205] = {X 234.4233, Y 102.1337, Z -6.3333, A 0.000, B 0.000, C 0.000 }
gfCNCPoint4[29206] = {X 233.4798, Y 102.2400, Z -6.3333, A 0.000, B 0.000, C 0.000 }
gfCNCPoint4[29207] = {X 214.1790, Y 102.2400, Z -6.3333, A 0.000, B 0.000, C 0.000 }
gfCNCPoint4[29208] = {X 213.7861, Y 102.2218, Z -6.3333, A 0.000, B 0.000, C 0.000 }
gfCNCPoint4[29209] = {X 213.3966, Y 102.1672, Z -6.3333, A 0.000, B 0.000, C 0.000 }
gfCNCPoint4[29210] = {X 213.0070, Y 102.2218, Z -6.3333, A 0.000, B 0.000, C 0.000 }
gfCNCPoint4[29211] = {X 212.6141, Y 102.2400, Z -6.3333, A 0.000, B 0.000, C 0.000 }
gfCNCPoint4[29212] = {X 194.9870, Y 102.2400, Z -6.3333, A 0.000, B 0.000, C 0.000 }
gfCNCPoint4[29213] = {X 194.0435, Y 102.1337, Z -6.3333, A 0.000, B 0.000, C 0.000 }
gfCNCPoint4[29214] = {X 193.1473, Y 101.8201, Z -6.3333, A 0.000, B 0.000, C 0.000 }
gfCNCPoint4[29215] = {X 192.3434, Y 101.3150, Z -6.3333, A 0.000, B 0.000, C 0.000 }
gfCNCPoint4[29216] = {X 191.6720, Y 100.6436, Z -6.3333, A 0.000, B 0.000, C 0.000 }
gfCNCPoint4[29217] = {X 191.1669, Y 99.8397, Z -6.3333, A 0.000, B 0.000, C 0.000 }
gfCNCPoint4[29218] = {X 190.8533, Y 98.9435, Z -6.3333, A 0.000, B 0.000, C 0.000 }
gfCNCPoint4[29219] = {X 190.7470, Y 98.0000, Z -6.3333, A 0.000, B 0.000, C 0.000 }
gfCNCPoint4[29220] = {X 190.7470, Y 97.0659, Z -6.3333, A 0.000, B 0.000, C 0.000 }
gfCNCPoint4[29221] = {X 190.8557, Y 96.1118, Z -6.3333, A 0.000, B 0.000, C 0.000 }
gfCNCPoint4[29222] = {X 191.1764, Y 95.2065, Z -6.3333, A 0.000, B 0.000, C 0.000 }
gfCNCPoint4[29223] = {X 191.6926, Y 94.3967, Z -6.3333, A 0.000, B 0.000, C 0.000 }
gfCNCPoint4[29224] = {X 188.5999, Y 91.0202, Z -6.3333, A 0.000, B 0.000, C 0.000 }
gfCNCPoint4[29225] = {X 150.0543, Y 91.0202, Z -6.3333, A 0.000, B 0.000, C 0.000 }
gfCNCPoint4[29226] = {X 147.0401, Y 94.3596, Z -6.3333, A 0.000, B 0.000, C 0.000 }
gfCNCPoint4[29227] = {X 147.5726, Y 95.1779, Z -6.3333, A 0.000, B 0.000, C 0.000 }
gfCNCPoint4[29228] = {X 147.9048, Y 96.0959, Z -6.3333, A 0.000, B 0.000, C 0.000 }
gfCNCPoint4[29229] = {X 148.0191, Y 97.0655, Z -6.3333, A 0.000, B 0.000, C 0.000 }
gfCNCPoint4[29230] = {X 148.0191, Y 98.0000, Z -6.3333, A 0.000, B 0.000, C 0.000 }
gfCNCPoint4[29231] = {X 147.9128, Y 98.9435, Z -6.3333, A 0.000, B 0.000, C 0.000 }
gfCNCPoint4[29232] = {X 147.5992, Y 99.8397, Z -6.3333, A 0.000, B 0.000, C 0.000 }
gfCNCPoint4[29233] = {X 147.0941, Y 100.6436, Z -6.3333, A 0.000, B 0.000, C 0.000 }
gfCNCPoint4[29234] = {X 146.4227, Y 101.3150, Z -6.3333, A 0.000, B 0.000, C 0.000 }
gfCNCPoint4[29235] = {X 145.6188, Y 101.8201, Z -6.3333, A 0.000, B 0.000, C 0.000 }
gfCNCPoint4[29236] = {X 144.7226, Y 102.1337, Z -6.3333, A 0.000, B 0.000, C 0.000 }
gfCNCPoint4[29237] = {X 143.7791, Y 102.2400, Z -6.3333, A 0.000, B 0.000, C 0.000 }
gfCNCPoint4[29238] = {X 125.0000, Y 102.2400, Z -6.3333, A 0.000, B 0.000, C 0.000 }
gfCNCPoint4[29239] = {X 124.0565, Y 102.1337, Z -6.3333, A 0.000, B 0.000, C 0.000 }
gfCNCPoint4[29240] = {X 123.1603, Y 101.8201, Z -6.3333, A 0.000, B 0.000, C 0.000 }
gfCNCPoint4[29241] = {X 122.3564, Y 101.3150, Z -6.3333, A 0.000, B 0.000, C 0.000 }
gfCNCPoint4[29242] = {X 121.6850, Y 100.6436, Z -6.3333, A 0.000, B 0.000, C 0.000 }
gfCNCPoint4[29243] = {X 121.1799, Y 99.8397, Z -6.3333, A 0.000, B 0.000, C 0.000 }
gfCNCPoint4[29244] = {X 120.8663, Y 98.9435, Z -6.3333, A 0.000, B 0.000, C 0.000 }
gfCNCPoint4[29245] = {X 120.7600, Y 98.0000, Z -6.3333, A 0.000, B 0.000, C 0.000 }
gfCNCPoint4[29246] = {X 120.7600, Y 97.0659, Z -6.3333, A 0.000, B 0.000, C 0.000 }
gfCNCPoint4[29247] = {X 120.8618, Y 96.1424, Z -6.3333, A 0.000, B 0.000, C 0.000 }
gfCNCPoint4[29248] = {X 121.1623, Y 95.2633, Z -6.3333, A 0.000, B 0.000, C 0.000 }
gfCNCPoint4[29249] = {X 121.6471, Y 94.4707, Z -6.3333, A 0.000, B 0.000, C 0.000 }
gfCNCPoint4[29250] = {X 122.2928, Y 93.8027, Z -6.3333, A 0.000, B 0.000, C 0.000 }
gfCNCPoint4[29251] = {X 123.0686, Y 93.2914, Z -6.3333, A 0.000, B 0.000, C 0.000 }
gfCNCPoint4[29252] = {X 123.9371, Y 92.9613, Z -6.3333, A 0.000, B 0.000, C 0.000 }
gfCNCPoint4[29253] = {X 124.8566, Y 92.8284, Z -6.3333, A 0.000, B 0.000, C 0.000 }
gfCNCPoint4[29254] = {X 124.8968, Y 92.8103, Z -6.3333, A 0.000, B 0.000, C 0.000 }
gfCNCPoint4[29255] = {X 124.9395, Y 92.7999, Z -6.3333, A 0.000, B 0.000, C 0.000 }
gfCNCPoint4[29256] = {X 125.4606, Y 92.7226, Z -6.3333, A 0.000, B 0.000, C 0.000 }
gfCNCPoint4[29257] = {X 126.3058, Y 92.5801, Z -6.3333, A 0.000, B 0.000, C 0.000 }
gfCNCPoint4[29258] = {X 127.1392, Y 92.3793, Z -6.3333, A 0.000, B 0.000, C 0.000 }
gfCNCPoint4[29259] = {X 128.3711, Y 91.2194, Z -6.3333, A 0.000, B 0.000, C 0.000 }
gfCNCPoint4[29260] = {X 129.5377, Y 89.9938, Z -6.3333, A 0.000, B 0.000, C 0.000 }
gfCNCPoint4[29261] = {X 140.7391, Y 77.6930, Z -6.3333, A 0.000, B 0.000, C 0.000 }
gfCNCPoint4[29262] = {X 137.7817, Y 74.9999, Z -6.3333, A 0.000, B 0.000, C 0.000 }
gfCNCPoint4[29263] = {X 140.7983, Y 77.7469, Z -6.3333, A 0.000, B 0.000, C 0.000 }
gfCNCPoint4[29264] = {X 155.8332, Y 61.2365, Z -6.3333, A 0.000, B 0.000, C 0.000 }
gfCNCPoint4[29265] = {X 155.4563, Y 60.5301, Z -6.3333, A 0.000, B 0.000, C 0.000 }
gfCNCPoint4[29266] = {X 155.2217, Y 59.7647, Z -6.3333, A 0.000, B 0.000, C 0.000 }
gfCNCPoint4[29267] = {X 155.1381, Y 58.9684, Z -6.3333, A 0.000, B 0.000, C 0.000 }
gfCNCPoint4[29268] = {X 155.1380, Y 58.0000, Z -6.3333, A 0.000, B 0.000, C 0.000 }
gfCNCPoint4[29269] = {X 155.2423, Y 57.0743, Z -6.3333, A 0.000, B 0.000, C 0.000 }
gfCNCPoint4[29270] = {X 155.5499, Y 56.1950, Z -6.3333, A 0.000, B 0.000, C 0.000 }
gfCNCPoint4[29271] = {X 156.0455, Y 55.4063, Z -6.3333, A 0.000, B 0.000, C 0.000 }
gfCNCPoint4[29272] = {X 156.7042, Y 54.7476, Z -6.3333, A 0.000, B 0.000, C 0.000 }
gfCNCPoint4[29273] = {X 157.4930, Y 54.2520, Z -6.3333, A 0.000, B 0.000, C 0.000 }
gfCNCPoint4[29274] = {X 158.3723, Y 53.9443, Z -6.3333, A 0.000, B 0.000, C 0.000 }
gfCNCPoint4[29275] = {X 159.2980, Y 53.8400, Z -6.3333, A 0.000, B 0.000, C 0.000 }
gfCNCPoint4[29276] = {X 178.5335, Y 53.8400, Z -6.3333, A 0.000, B 0.000, C 0.000 }
gfCNCPoint4[29277] = {X 179.4592, Y 53.9443, Z -6.3333, A 0.000, B 0.000, C 0.000 }
gfCNCPoint4[29278] = {X 180.3385, Y 54.2520, Z -6.3333, A 0.000, B 0.000, C 0.000 }
gfCNCPoint4[29279] = {X 181.1272, Y 54.7476, Z -6.3333, A 0.000, B 0.000, C 0.000 }
gfCNCPoint4[29280] = {X 181.7859, Y 55.4063, Z -6.3333, A 0.000, B 0.000, C 0.000 }
gfCNCPoint4[29281] = {X 182.2815, Y 56.1950, Z -6.3333, A 0.000, B 0.000, C 0.000 }
gfCNCPoint4[29282] = {X 182.5892, Y 57.0743, Z -6.3333, A 0.000, B 0.000, C 0.000 }
gfCNCPoint4[29283] = {X 182.6935, Y 58.0000, Z -6.3333, A 0.000, B 0.000, C 0.000 }
gfCNCPoint4[29284] = {X 182.6935, Y 58.9342, Z -6.3333, A 0.000, B 0.000, C 0.000 }
gfCNCPoint4[29285] = {X 182.6160, Y 59.7333, Z -6.3333, A 0.000, B 0.000, C 0.000 }
gfCNCPoint4[29286] = {X 182.3865, Y 60.5025, Z -6.3333, A 0.000, B 0.000, C 0.000 }
gfCNCPoint4[29287] = {X 182.0135, Y 61.2134, Z -6.3333, A 0.000, B 0.000, C 0.000 }
gfCNCPoint4[29288] = {X 209.3617, Y 91.0624, Z -6.3333, A 0.000, B 0.000, C 0.000 }
gfCNCPoint4[29289] = {X 210.0263, Y 91.7368, Z -6.3333, A 0.000, B 0.000, C 0.000 }
gfCNCPoint4[29290] = {X 210.7382, Y 92.3609, Z -6.3333, A 0.000, B 0.000, C 0.000 }
gfCNCPoint4[29291] = {X 211.0466, Y 92.5558, Z -6.3333, A 0.000, B 0.000, C 0.000 }
gfCNCPoint4[29292] = {X 211.3925, Y 92.6720, Z -6.3333, A 0.000, B 0.000, C 0.000 }
gfCNCPoint4[29293] = {X 213.3995, Y 92.9851, Z -6.3333, A 0.000, B 0.000, C 0.000 }
gfCNCPoint4[29294] = {X 214.4547, Y 92.8955, Z -6.3333, A 0.000, B 0.000, C 0.000 }
gfCNCPoint4[29295] = {X 215.5121, Y 92.8348, Z -6.3333, A 0.000, B 0.000, C 0.000 }
gfCNCPoint4[29296] = {X 216.2109, Y 92.7583, Z -6.3333, A 0.000, B 0.000, C 0.000 }
gfCNCPoint4[29297] = {X 216.8837, Y 92.5547, Z -6.3333, A 0.000, B 0.000, C 0.000 }
gfCNCPoint4[29298] = {X 217.5077, Y 92.2309, Z -6.3333, A 0.000, B 0.000, C 0.000 }
gfCNCPoint4[29299] = {X 223.0478, Y 88.6556, Z -6.3333, A 0.000, B 0.000, C 0.000 }
gfCNCPoint4[29300] = {X 246.1781, Y 73.8653, Z -6.3333, A 0.000, B 0.000, C 0.000 }
gfCNCPoint4[29301] = {X 221.6899, Y 64.2558, Z -6.3333, A 0.000, B 0.000, C 0.000 }
gfCNCPoint4[29302] = {X 219.9051, Y 63.6585, Z -6.3333, A 0.000, B 0.000, C 0.000 }
gfCNCPoint4[29303] = {X 218.0638, Y 63.2687, Z -6.3333, A 0.000, B 0.000, C 0.000 }
gfCNCPoint4[29304] = {X 216.1900, Y 63.0917, Z -6.3333, A 0.000, B 0.000, C 0.000 }
gfCNCPoint4[29305] = {X 215.2926, Y 62.9624, Z -6.3333, A 0.000, B 0.000, C 0.000 }
gfCNCPoint4[29306] = {X 214.4445, Y 62.6418, Z -6.3333, A 0.000, B 0.000, C 0.000 }
gfCNCPoint4[29307] = {X 213.6860, Y 62.1451, Z -6.3333, A 0.000, B 0.000, C 0.000 }
gfCNCPoint4[29308] = {X 213.0531, Y 61.4958, Z -6.3333, A 0.000, B 0.000, C 0.000 }
gfCNCPoint4[29309] = {X 212.5760, Y 60.7249, Z -6.3333, A 0.000, B 0.000, C 0.000 }
gfCNCPoint4[29310] = {X 212.2772, Y 59.8688, Z -6.3333, A 0.000, B 0.000, C 0.000 }
gfCNCPoint4[29311] = {X 212.1710, Y 58.9684, Z -6.3333, A 0.000, B 0.000, C 0.000 }
gfCNCPoint4[29312] = {X 212.1708, Y 58.0000, Z -6.3333, A 0.000, B 0.000, C 0.000 }
gfCNCPoint4[29313] = {X 212.2751, Y 57.0743, Z -6.3333, A 0.000, B 0.000, C 0.000 }
gfCNCPoint4[29314] = {X 212.5828, Y 56.1950, Z -6.3333, A 0.000, B 0.000, C 0.000 }
gfCNCPoint4[29315] = {X 213.0784, Y 55.4063, Z -6.3333, A 0.000, B 0.000, C 0.000 }
gfCNCPoint4[29316] = {X 213.7371, Y 54.7476, Z -6.3333, A 0.000, B 0.000, C 0.000 }
gfCNCPoint4[29317] = {X 214.5259, Y 54.2520, Z -6.3333, A 0.000, B 0.000, C 0.000 }
gfCNCPoint4[29318] = {X 215.4051, Y 53.9443, Z -6.3333, A 0.000, B 0.000, C 0.000 }
gfCNCPoint4[29319] = {X 216.3308, Y 53.8400, Z -6.3333, A 0.000, B 0.000, C 0.000 }
gfCNCPoint4[29320] = {X 237.2617, Y 53.8400, Z -6.3333, A 0.000, B 0.000, C 0.000 }
gfCNCPoint4[29321] = {X 238.1874, Y 53.9443, Z -6.3333, A 0.000, B 0.000, C 0.000 }
gfCNCPoint4[29322] = {X 239.0666, Y 54.2520, Z -6.3333, A 0.000, B 0.000, C 0.000 }
gfCNCPoint4[29323] = {X 239.8554, Y 54.7476, Z -6.3333, A 0.000, B 0.000, C 0.000 }
gfCNCPoint4[29324] = {X 240.5141, Y 55.4063, Z -6.3333, A 0.000, B 0.000, C 0.000 }
gfCNCPoint4[29325] = {X 241.0097, Y 56.1950, Z -6.3333, A 0.000, B 0.000, C 0.000 }
gfCNCPoint4[29326] = {X 241.3174, Y 57.0743, Z -6.3333, A 0.000, B 0.000, C 0.000 }
gfCNCPoint4[29327] = {X 241.4217, Y 58.0000, Z -6.3333, A 0.000, B 0.000, C 0.000 }
gfCNCPoint4[29328] = {X 241.4217, Y 58.3413, Z -6.3333, A 0.000, B 0.000, C 0.000 }
gfCNCPoint4[29329] = {X 248.0559, Y 60.9282, Z -6.3333, A 0.000, B 0.000, C 0.000 }
gfCNCPoint4[29330] = {X 275.7922, Y 71.9372, Z -6.3333, A 0.000, B 0.000, C 0.000 }
gfCNCPoint4[29331] = {X 275.7937, Y 63.0708, Z -6.3333, A 0.000, B 0.000, C 0.000 }
gfCNCPoint4[29332] = {X 275.6911, Y 63.0587, Z -6.3333, A 0.000, B 0.000, C 0.000 }
gfCNCPoint4[29333] = {X 275.5889, Y 63.0440, Z -6.3333, A 0.000, B 0.000, C 0.000 }
gfCNCPoint4[29334] = {X 274.6515, Y 62.7818, Z -6.3333, A 0.000, B 0.000, C 0.000 }
gfCNCPoint4[29335] = {X 273.8006, Y 62.3091, Z -6.3333, A 0.000, B 0.000, C 0.000 }
gfCNCPoint4[29336] = {X 273.0829, Y 61.6515, Z -6.3333, A 0.000, B 0.000, C 0.000 }
gfCNCPoint4[29337] = {X 272.5376, Y 60.8451, Z -6.3333, A 0.000, B 0.000, C 0.000 }
gfCNCPoint4[29338] = {X 272.1947, Y 59.9342, Z -6.3333, A 0.000, B 0.000, C 0.000 }
gfCNCPoint4[29339] = {X 272.0728, Y 58.9684, Z -6.3333, A 0.000, B 0.000, C 0.000 }
gfCNCPoint4[29340] = {X 272.0727, Y 58.0000, Z -6.3333, A 0.000, B 0.000, C 0.000 }
gfCNCPoint4[29341] = {X 272.1770, Y 57.0743, Z -6.3333, A 0.000, B 0.000, C 0.000 }
gfCNCPoint4[29342] = {X 272.4847, Y 56.1950, Z -6.3333, A 0.000, B 0.000, C 0.000 }
gfCNCPoint4[29343] = {X 272.9803, Y 55.4063, Z -6.3333, A 0.000, B 0.000, C 0.000 }
gfCNCPoint4[29344] = {X 273.6390, Y 54.7476, Z -6.3333, A 0.000, B 0.000, C 0.000 }
gfCNCPoint4[29345] = {X 274.4277, Y 54.2520, Z -6.3333, A 0.000, B 0.000, C 0.000 }
gfCNCPoint4[29346] = {X 275.3070, Y 53.9443, Z -6.3333, A 0.000, B 0.000, C 0.000 }
gfCNCPoint4[29347] = {X 276.2327, Y 53.8400, Z -6.3333, A 0.000, B 0.000, C 0.000 }
gfCNCPoint4[29348] = {X 292.7731, Y 53.8400, Z -6.3333, A 0.000, B 0.000, C 0.000 }
gfCNCPoint4[29349] = {X 293.6988, Y 53.9443, Z -6.3333, A 0.000, B 0.000, C 0.000 }
gfCNCPoint4[29350] = {X 294.5780, Y 54.2520, Z -6.3333, A 0.000, B 0.000, C 0.000 }
gfCNCPoint4[29351] = {X 295.3668, Y 54.7476, Z -6.3333, A 0.000, B 0.000, C 0.000 }
gfCNCPoint4[29352] = {X 296.0255, Y 55.4063, Z -6.3333, A 0.000, B 0.000, C 0.000 }
gfCNCPoint4[29353] = {X 296.5211, Y 56.1950, Z -6.3333, A 0.000, B 0.000, C 0.000 }
gfCNCPoint4[29354] = {X 296.8288, Y 57.0743, Z -6.3333, A 0.000, B 0.000, C 0.000 }
gfCNCPoint4[29355] = {X 296.9331, Y 58.0000, Z -6.3333, A 0.000, B 0.000, C 0.000 }
gfCNCPoint4[29356] = {X 296.9331, Y 58.9346, Z -6.3333, A 0.000, B 0.000, C 0.000 }
gfCNCPoint4[29357] = {X 296.8156, Y 59.9063, Z -6.3333, A 0.000, B 0.000, C 0.000 }
gfCNCPoint4[29358] = {X 296.4751, Y 60.8240, Z -6.3333, A 0.000, B 0.000, C 0.000 }
gfCNCPoint4[29359] = {X 295.9304, Y 61.6373, Z -6.3333, A 0.000, B 0.000, C 0.000 }
gfCNCPoint4[29360] = {X 295.2113, Y 62.3014, Z -6.3333, A 0.000, B 0.000, C 0.000 }
gfCNCPoint4[29361] = {X 294.3574, Y 62.7799, Z -6.3333, A 0.000, B 0.000, C 0.000 }
gfCNCPoint4[29362] = {X 293.4156, Y 63.0465, Z -6.3333, A 0.000, B 0.000, C 0.000 }
gfCNCPoint4[29363] = {X 293.3189, Y 63.0608, Z -6.3333, A 0.000, B 0.000, C 0.000 }
gfCNCPoint4[29364] = {X 293.2219, Y 63.0728, Z -6.3333, A 0.000, B 0.000, C 0.000 }
gfCNCPoint4[29365] = {X 293.2134, Y 63.1616, Z -6.3333, A 0.000, B 0.000, C 0.000 }
gfCNCPoint4[29366] = {X 293.2248, Y 92.9206, Z -6.3333, A 0.000, B 0.000, C 0.000 }
gfCNCPoint4[29367] = {X 293.3200, Y 92.9328, Z -6.3333, A 0.000, B 0.000, C 0.000 }
gfCNCPoint4[29368] = {X 293.4148, Y 92.9471, Z -6.3333, A 0.000, B 0.000, C 0.000 }
gfCNCPoint4[29369] = {X 294.3563, Y 93.2164, Z -6.3333, A 0.000, B 0.000, C 0.000 }
gfCNCPoint4[29370] = {X 295.2096, Y 93.6967, Z -6.3333, A 0.000, B 0.000, C 0.000 }
gfCNCPoint4[29371] = {X 295.9282, Y 94.3618, Z -6.3333, A 0.000, B 0.000, C 0.000 }
gfCNCPoint4[29372] = {X 296.4730, Y 95.1755, Z -6.3333, A 0.000, B 0.000, C 0.000 }
gfCNCPoint4[29373] = {X 296.8141, Y 96.0933, Z -6.3333, A 0.000, B 0.000, C 0.000 }
gfCNCPoint4[29374] = {X 296.9331, Y 97.0653, Z -6.3333, A 0.000, B 0.000, C 0.000 }
gfCNCPoint4[29375] = {X 296.9331, Y 98.0000, Z -6.3333, A 0.000, B 0.000, C 0.000 }
gfCNCPoint4[29376] = {X 296.8288, Y 98.9257, Z -6.3333, A 0.000, B 0.000, C 0.000 }
gfCNCPoint4[29377] = {X 296.5211, Y 99.8050, Z -6.3333, A 0.000, B 0.000, C 0.000 }
gfCNCPoint4[29378] = {X 296.0255, Y 100.5937, Z -6.3333, A 0.000, B 0.000, C 0.000 }
gfCNCPoint4[29379] = {X 295.3668, Y 101.2524, Z -6.3333, A 0.000, B 0.000, C 0.000 }
gfCNCPoint4[29380] = {X 294.5780, Y 101.7480, Z -6.3333, A 0.000, B 0.000, C 0.000 }
gfCNCPoint4[29381] = {X 293.6988, Y 102.0557, Z -6.3333, A 0.000, B 0.000, C 0.000 }
gfCNCPoint4[29382] = {X 292.7731, Y 102.1600, Z -6.3333, A 0.000, B 0.000, C 0.000 }
gfCNCPoint4[29383] = {X 276.2327, Y 102.1600, Z -6.3333, A 0.000, B 0.000, C 0.000 }
gfCNCPoint4[29384] = {X 275.3070, Y 102.0557, Z -6.3333, A 0.000, B 0.000, C 0.000 }
gfCNCPoint4[29385] = {X 274.4277, Y 101.7480, Z -6.3333, A 0.000, B 0.000, C 0.000 }
gfCNCPoint4[29386] = {X 273.6390, Y 101.2524, Z -6.3333, A 0.000, B 0.000, C 0.000 }
gfCNCPoint4[29387] = {X 272.9803, Y 100.5937, Z -6.3333, A 0.000, B 0.000, C 0.000 }
gfCNCPoint4[29388] = {X 272.4847, Y 99.8050, Z -6.3333, A 0.000, B 0.000, C 0.000 }
gfCNCPoint4[29389] = {X 272.1770, Y 98.9257, Z -6.3333, A 0.000, B 0.000, C 0.000 }
gfCNCPoint4[29390] = {X 272.0727, Y 98.0000, Z -6.3333, A 0.000, B 0.000, C 0.000 }
gfCNCPoint4[29391] = {X 272.0727, Y 97.0659, Z -6.3333, A 0.000, B 0.000, C 0.000 }
gfCNCPoint4[29392] = {X 272.1634, Y 96.2021, Z -6.3333, A 0.000, B 0.000, C 0.000 }
gfCNCPoint4[29393] = {X 272.4314, Y 95.3761, Z -6.3333, A 0.000, B 0.000, C 0.000 }
gfCNCPoint4[29394] = {X 272.8651, Y 94.6237, Z -6.3333, A 0.000, B 0.000, C 0.000 }
gfCNCPoint4[29395] = {X 273.4455, Y 93.9777, Z -6.3333, A 0.000, B 0.000, C 0.000 }
gfCNCPoint4[29396] = {X 274.1474, Y 93.4663, Z -6.3333, A 0.000, B 0.000, C 0.000 }
gfCNCPoint4[29397] = {X 274.9403, Y 93.1118, Z -6.3333, A 0.000, B 0.000, C 0.000 }
gfCNCPoint4[29398] = {X 275.7894, Y 92.9296, Z -6.3333, A 0.000, B 0.000, C 0.000 }
gfCNCPoint4[29399] = {X 275.7894, Y 85.4858, Z -6.3333, A 0.000, B 0.000, C 0.000 }
gfCNCPoint4[29400] = {X 262.6228, Y 80.3245, Z -6.3333, A 0.000, B 0.000, C 0.000 }
gfCNCPoint4[29401] = {X 262.1916, Y 80.5967, Z -6.3333, A 0.000, B 0.000, C 0.000 }
gfCNCPoint4[29402] = {X 237.6367, Y 96.5016, Z -6.3333, A 0.000, B 0.000, C 0.000 }
gfCNCPoint4[29403] = {X 237.6398, Y 97.0655, Z -6.3333, A 0.000, B 0.000, C 0.000 }
gfCNCPoint4[29404] = {X 237.6398, Y 98.0000, Z -6.3333, A 0.000, B 0.000, C 0.000 }
gfCNCPoint4[29405] = {X 237.5355, Y 98.9257, Z -6.3333, A 0.000, B 0.000, C 0.000 }
gfCNCPoint4[29406] = {X 237.2278, Y 99.8050, Z -6.3333, A 0.000, B 0.000, C 0.000 }
gfCNCPoint4[29407] = {X 236.7322, Y 100.5937, Z -6.3333, A 0.000, B 0.000, C 0.000 }
gfCNCPoint4[29408] = {X 236.0735, Y 101.2524, Z -6.3333, A 0.000, B 0.000, C 0.000 }
gfCNCPoint4[29409] = {X 235.2847, Y 101.7480, Z -6.3333, A 0.000, B 0.000, C 0.000 }
gfCNCPoint4[29410] = {X 234.4055, Y 102.0557, Z -6.3333, A 0.000, B 0.000, C 0.000 }
gfCNCPoint4[29411] = {X 233.4798, Y 102.1600, Z -6.3333, A 0.000, B 0.000, C 0.000 }
gfCNCPoint4[29412] = {X 214.1790, Y 102.1600, Z -6.3333, A 0.000, B 0.000, C 0.000 }
gfCNCPoint4[29413] = {X 213.7860, Y 102.1414, Z -6.3333, A 0.000, B 0.000, C 0.000 }
gfCNCPoint4[29414] = {X 213.3966, Y 102.0857, Z -6.3333, A 0.000, B 0.000, C 0.000 }
gfCNCPoint4[29415] = {X 213.0071, Y 102.1414, Z -6.3333, A 0.000, B 0.000, C 0.000 }
gfCNCPoint4[29416] = {X 212.6141, Y 102.1600, Z -6.3333, A 0.000, B 0.000, C 0.000 }
gfCNCPoint4[29417] = {X 194.9870, Y 102.1600, Z -6.3333, A 0.000, B 0.000, C 0.000 }
gfCNCPoint4[29418] = {X 194.0613, Y 102.0557, Z -6.3333, A 0.000, B 0.000, C 0.000 }
gfCNCPoint4[29419] = {X 193.1820, Y 101.7480, Z -6.3333, A 0.000, B 0.000, C 0.000 }
gfCNCPoint4[29420] = {X 192.3932, Y 101.2524, Z -6.3333, A 0.000, B 0.000, C 0.000 }
gfCNCPoint4[29421] = {X 191.7345, Y 100.5937, Z -6.3333, A 0.000, B 0.000, C 0.000 }
gfCNCPoint4[29422] = {X 191.2389, Y 99.8050, Z -6.3333, A 0.000, B 0.000, C 0.000 }
gfCNCPoint4[29423] = {X 190.9313, Y 98.9257, Z -6.3333, A 0.000, B 0.000, C 0.000 }
gfCNCPoint4[29424] = {X 190.8270, Y 98.0000, Z -6.3333, A 0.000, B 0.000, C 0.000 }
gfCNCPoint4[29425] = {X 190.8270, Y 97.0659, Z -6.3333, A 0.000, B 0.000, C 0.000 }
gfCNCPoint4[29426] = {X 190.9241, Y 96.1723, Z -6.3333, A 0.000, B 0.000, C 0.000 }
gfCNCPoint4[29427] = {X 191.2109, Y 95.3203, Z -6.3333, A 0.000, B 0.000, C 0.000 }
gfCNCPoint4[29428] = {X 191.6741, Y 94.5499, Z -6.3333, A 0.000, B 0.000, C 0.000 }
gfCNCPoint4[29429] = {X 191.7354, Y 94.4712, Z -6.3333, A 0.000, B 0.000, C 0.000 }
gfCNCPoint4[29430] = {X 191.7986, Y 94.3939, Z -6.3333, A 0.000, B 0.000, C 0.000 }
gfCNCPoint4[29431] = {X 188.6351, Y 90.9402, Z -6.3333, A 0.000, B 0.000, C 0.000 }
gfCNCPoint4[29432] = {X 150.0187, Y 90.9402, Z -6.3333, A 0.000, B 0.000, C 0.000 }
gfCNCPoint4[29433] = {X 146.9339, Y 94.3578, Z -6.3333, A 0.000, B 0.000, C 0.000 }
gfCNCPoint4[29434] = {X 147.4802, Y 95.1724, Z -6.3333, A 0.000, B 0.000, C 0.000 }
gfCNCPoint4[29435] = {X 147.8216, Y 96.0919, Z -6.3333, A 0.000, B 0.000, C 0.000 }
gfCNCPoint4[29436] = {X 147.9391, Y 97.0657, Z -6.3333, A 0.000, B 0.000, C 0.000 }
gfCNCPoint4[29437] = {X 147.9391, Y 98.0000, Z -6.3333, A 0.000, B 0.000, C 0.000 }
gfCNCPoint4[29438] = {X 147.8348, Y 98.9257, Z -6.3333, A 0.000, B 0.000, C 0.000 }
gfCNCPoint4[29439] = {X 147.5271, Y 99.8050, Z -6.3333, A 0.000, B 0.000, C 0.000 }
gfCNCPoint4[29440] = {X 147.0315, Y 100.5937, Z -6.3333, A 0.000, B 0.000, C 0.000 }
gfCNCPoint4[29441] = {X 146.3728, Y 101.2524, Z -6.3333, A 0.000, B 0.000, C 0.000 }
gfCNCPoint4[29442] = {X 145.5841, Y 101.7480, Z -6.3333, A 0.000, B 0.000, C 0.000 }
gfCNCPoint4[29443] = {X 144.7048, Y 102.0557, Z -6.3333, A 0.000, B 0.000, C 0.000 }
gfCNCPoint4[29444] = {X 143.7791, Y 102.1600, Z -6.3333, A 0.000, B 0.000, C 0.000 }
gfCNCPoint4[29445] = {X 125.0000, Y 102.1600, Z -6.3333, A 0.000, B 0.000, C 0.000 }
gfCNCPoint4[29446] = {X 124.0743, Y 102.0557, Z -6.3333, A 0.000, B 0.000, C 0.000 }
gfCNCPoint4[29447] = {X 123.1950, Y 101.7480, Z -6.3333, A 0.000, B 0.000, C 0.000 }
gfCNCPoint4[29448] = {X 122.4063, Y 101.2524, Z -6.3333, A 0.000, B 0.000, C 0.000 }
gfCNCPoint4[29449] = {X 121.7476, Y 100.5937, Z -6.3333, A 0.000, B 0.000, C 0.000 }
gfCNCPoint4[29450] = {X 121.2520, Y 99.8050, Z -6.3333, A 0.000, B 0.000, C 0.000 }
gfCNCPoint4[29451] = {X 120.9443, Y 98.9257, Z -6.3333, A 0.000, B 0.000, C 0.000 }
gfCNCPoint4[29452] = {X 120.8400, Y 98.0000, Z -6.3333, A 0.000, B 0.000, C 0.000 }
gfCNCPoint4[29453] = {X 120.8400, Y 97.0659, Z -6.3333, A 0.000, B 0.000, C 0.000 }
gfCNCPoint4[29454] = {X 120.9405, Y 96.1568, Z -6.3333, A 0.000, B 0.000, C 0.000 }
gfCNCPoint4[29455] = {X 121.2373, Y 95.2917, Z -6.3333, A 0.000, B 0.000, C 0.000 }
gfCNCPoint4[29456] = {X 121.7160, Y 94.5123, Z -6.3333, A 0.000, B 0.000, C 0.000 }
gfCNCPoint4[29457] = {X 122.3534, Y 93.8564, Z -6.3333, A 0.000, B 0.000, C 0.000 }
gfCNCPoint4[29458] = {X 123.1188, Y 93.3556, Z -6.3333, A 0.000, B 0.000, C 0.000 }
gfCNCPoint4[29459] = {X 123.9751, Y 93.0342, Z -6.3333, A 0.000, B 0.000, C 0.000 }
gfCNCPoint4[29460] = {X 124.8809, Y 92.9076, Z -6.3333, A 0.000, B 0.000, C 0.000 }
gfCNCPoint4[29461] = {X 124.9144, Y 92.8891, Z -6.3333, A 0.000, B 0.000, C 0.000 }
gfCNCPoint4[29462] = {X 124.9512, Y 92.8791, Z -6.3333, A 0.000, B 0.000, C 0.000 }
gfCNCPoint4[29463] = {X 125.4717, Y 92.8019, Z -6.3333, A 0.000, B 0.000, C 0.000 }
gfCNCPoint4[29464] = {X 126.3313, Y 92.6565, Z -6.3333, A 0.000, B 0.000, C 0.000 }
gfCNCPoint4[29465] = {X 127.1785, Y 92.4514, Z -6.3333, A 0.000, B 0.000, C 0.000 }
gfCNCPoint4[29466] = {X 128.4210, Y 91.2827, Z -6.3333, A 0.000, B 0.000, C 0.000 }
gfCNCPoint4[29467] = {X 129.5971, Y 90.0473, Z -6.3333, A 0.000, B 0.000, C 0.000 }
gfCNCPoint4[29468] = {X 140.7983, Y 77.7469, Z -6.3333, A 0.000, B 0.000, C 0.000 }
gfCNCPoint4[29469] = {X 137.8408, Y 75.0537, Z -6.3333, A 0.000, B 0.000, C 0.000 }
gfCNCPoint4[29470] = {X 140.8574, Y 77.8008, Z -6.3333, A 0.000, B 0.000, C 0.000 }
gfCNCPoint4[29471] = {X 155.9347, Y 61.2438, Z -6.3333, A 0.000, B 0.000, C 0.000 }
gfCNCPoint4[29472] = {X 155.5463, Y 60.5377, Z -6.3333, A 0.000, B 0.000, C 0.000 }
gfCNCPoint4[29473] = {X 155.3043, Y 59.7690, Z -6.3333, A 0.000, B 0.000, C 0.000 }
gfCNCPoint4[29474] = {X 155.2181, Y 58.9678, Z -6.3333, A 0.000, B 0.000, C 0.000 }
gfCNCPoint4[29475] = {X 155.2180, Y 58.0000, Z -6.3333, A 0.000, B 0.000, C 0.000 }
gfCNCPoint4[29476] = {X 155.3203, Y 57.0921, Z -6.3333, A 0.000, B 0.000, C 0.000 }
gfCNCPoint4[29477] = {X 155.6220, Y 56.2298, Z -6.3333, A 0.000, B 0.000, C 0.000 }
gfCNCPoint4[29478] = {X 156.1081, Y 55.4562, Z -6.3333, A 0.000, B 0.000, C 0.000 }
gfCNCPoint4[29479] = {X 156.7541, Y 54.8101, Z -6.3333, A 0.000, B 0.000, C 0.000 }
gfCNCPoint4[29480] = {X 157.5277, Y 54.3240, Z -6.3333, A 0.000, B 0.000, C 0.000 }
gfCNCPoint4[29481] = {X 158.3901, Y 54.0223, Z -6.3333, A 0.000, B 0.000, C 0.000 }
gfCNCPoint4[29482] = {X 159.2980, Y 53.9200, Z -6.3333, A 0.000, B 0.000, C 0.000 }
gfCNCPoint4[29483] = {X 178.5335, Y 53.9200, Z -6.3333, A 0.000, B 0.000, C 0.000 }
gfCNCPoint4[29484] = {X 179.4414, Y 54.0223, Z -6.3333, A 0.000, B 0.000, C 0.000 }
gfCNCPoint4[29485] = {X 180.3037, Y 54.3240, Z -6.3333, A 0.000, B 0.000, C 0.000 }
gfCNCPoint4[29486] = {X 181.0773, Y 54.8101, Z -6.3333, A 0.000, B 0.000, C 0.000 }
gfCNCPoint4[29487] = {X 181.7234, Y 55.4562, Z -6.3333, A 0.000, B 0.000, C 0.000 }
gfCNCPoint4[29488] = {X 182.2095, Y 56.2298, Z -6.3333, A 0.000, B 0.000, C 0.000 }
gfCNCPoint4[29489] = {X 182.5112, Y 57.0921, Z -6.3333, A 0.000, B 0.000, C 0.000 }
gfCNCPoint4[29490] = {X 182.6135, Y 58.0000, Z -6.3333, A 0.000, B 0.000, C 0.000 }
gfCNCPoint4[29491] = {X 182.6135, Y 58.9342, Z -6.3333, A 0.000, B 0.000, C 0.000 }
gfCNCPoint4[29492] = {X 182.5335, Y 59.7382, Z -6.3333, A 0.000, B 0.000, C 0.000 }
gfCNCPoint4[29493] = {X 182.2966, Y 60.5106, Z -6.3333, A 0.000, B 0.000, C 0.000 }
gfCNCPoint4[29494] = {X 181.9122, Y 61.2212, Z -6.3333, A 0.000, B 0.000, C 0.000 }
gfCNCPoint4[29495] = {X 209.3027, Y 91.1165, Z -6.3333, A 0.000, B 0.000, C 0.000 }
gfCNCPoint4[29496] = {X 209.9714, Y 91.7950, Z -6.3333, A 0.000, B 0.000, C 0.000 }
gfCNCPoint4[29497] = {X 210.6877, Y 92.4230, Z -6.3333, A 0.000, B 0.000, C 0.000 }
gfCNCPoint4[29498] = {X 211.0132, Y 92.6285, Z -6.3333, A 0.000, B 0.000, C 0.000 }
gfCNCPoint4[29499] = {X 211.3782, Y 92.7508, Z -6.3333, A 0.000, B 0.000, C 0.000 }
gfCNCPoint4[29500] = {X 213.3972, Y 93.0657, Z -6.3333, A 0.000, B 0.000, C 0.000 }
gfCNCPoint4[29501] = {X 214.4548, Y 92.9757, Z -6.3333, A 0.000, B 0.000, C 0.000 }
gfCNCPoint4[29502] = {X 215.5145, Y 92.9148, Z -6.3333, A 0.000, B 0.000, C 0.000 }
gfCNCPoint4[29503] = {X 216.2277, Y 92.8365, Z -6.3333, A 0.000, B 0.000, C 0.000 }
gfCNCPoint4[29504] = {X 216.9143, Y 92.6286, Z -6.3333, A 0.000, B 0.000, C 0.000 }
gfCNCPoint4[29505] = {X 217.5511, Y 92.2981, Z -6.3333, A 0.000, B 0.000, C 0.000 }
gfCNCPoint4[29506] = {X 223.0910, Y 88.7229, Z -6.3333, A 0.000, B 0.000, C 0.000 }
gfCNCPoint4[29507] = {X 246.3534, Y 73.8482, Z -6.3333, A 0.000, B 0.000, C 0.000 }
gfCNCPoint4[29508] = {X 221.7196, Y 64.1815, Z -6.3333, A 0.000, B 0.000, C 0.000 }
gfCNCPoint4[29509] = {X 219.9261, Y 63.5813, Z -6.3333, A 0.000, B 0.000, C 0.000 }
gfCNCPoint4[29510] = {X 218.0758, Y 63.1896, Z -6.3333, A 0.000, B 0.000, C 0.000 }
gfCNCPoint4[29511] = {X 216.1929, Y 63.0117, Z -6.3333, A 0.000, B 0.000, C 0.000 }
gfCNCPoint4[29512] = {X 215.3127, Y 62.8850, Z -6.3333, A 0.000, B 0.000, C 0.000 }
gfCNCPoint4[29513] = {X 214.4809, Y 62.5706, Z -6.3333, A 0.000, B 0.000, C 0.000 }
gfCNCPoint4[29514] = {X 213.7369, Y 62.0834, Z -6.3333, A 0.000, B 0.000, C 0.000 }
gfCNCPoint4[29515] = {X 213.1162, Y 61.4466, Z -6.3333, A 0.000, B 0.000, C 0.000 }
gfCNCPoint4[29516] = {X 212.6482, Y 60.6905, Z -6.3333, A 0.000, B 0.000, C 0.000 }
gfCNCPoint4[29517] = {X 212.3552, Y 59.8509, Z -6.3333, A 0.000, B 0.000, C 0.000 }
gfCNCPoint4[29518] = {X 212.2509, Y 58.9678, Z -6.3333, A 0.000, B 0.000, C 0.000 }
gfCNCPoint4[29519] = {X 212.2508, Y 58.0000, Z -6.3333, A 0.000, B 0.000, C 0.000 }
gfCNCPoint4[29520] = {X 212.3531, Y 57.0921, Z -6.3333, A 0.000, B 0.000, C 0.000 }
gfCNCPoint4[29521] = {X 212.6549, Y 56.2298, Z -6.3333, A 0.000, B 0.000, C 0.000 }
gfCNCPoint4[29522] = {X 213.1409, Y 55.4562, Z -6.3333, A 0.000, B 0.000, C 0.000 }
gfCNCPoint4[29523] = {X 213.7870, Y 54.8101, Z -6.3333, A 0.000, B 0.000, C 0.000 }
gfCNCPoint4[29524] = {X 214.5606, Y 54.3240, Z -6.3333, A 0.000, B 0.000, C 0.000 }
gfCNCPoint4[29525] = {X 215.4229, Y 54.0223, Z -6.3333, A 0.000, B 0.000, C 0.000 }
gfCNCPoint4[29526] = {X 216.3308, Y 53.9200, Z -6.3333, A 0.000, B 0.000, C 0.000 }
gfCNCPoint4[29527] = {X 237.2617, Y 53.9200, Z -6.3333, A 0.000, B 0.000, C 0.000 }
gfCNCPoint4[29528] = {X 238.1696, Y 54.0223, Z -6.3333, A 0.000, B 0.000, C 0.000 }
gfCNCPoint4[29529] = {X 239.0319, Y 54.3240, Z -6.3333, A 0.000, B 0.000, C 0.000 }
gfCNCPoint4[29530] = {X 239.8055, Y 54.8101, Z -6.3333, A 0.000, B 0.000, C 0.000 }
gfCNCPoint4[29531] = {X 240.4516, Y 55.4562, Z -6.3333, A 0.000, B 0.000, C 0.000 }
gfCNCPoint4[29532] = {X 240.9376, Y 56.2298, Z -6.3333, A 0.000, B 0.000, C 0.000 }
gfCNCPoint4[29533] = {X 241.2394, Y 57.0921, Z -6.3333, A 0.000, B 0.000, C 0.000 }
gfCNCPoint4[29534] = {X 241.3417, Y 58.0000, Z -6.3333, A 0.000, B 0.000, C 0.000 }
gfCNCPoint4[29535] = {X 241.3417, Y 58.3959, Z -6.3333, A 0.000, B 0.000, C 0.000 }
gfCNCPoint4[29536] = {X 248.0266, Y 61.0026, Z -6.3333, A 0.000, B 0.000, C 0.000 }
gfCNCPoint4[29537] = {X 275.8722, Y 72.0551, Z -6.3333, A 0.000, B 0.000, C 0.000 }
gfCNCPoint4[29538] = {X 275.8737, Y 62.9982, Z -6.3333, A 0.000, B 0.000, C 0.000 }
gfCNCPoint4[29539] = {X 275.7372, Y 62.9839, Z -6.3333, A 0.000, B 0.000, C 0.000 }
gfCNCPoint4[29540] = {X 275.6013, Y 62.9649, Z -6.3333, A 0.000, B 0.000, C 0.000 }
gfCNCPoint4[29541] = {X 274.6819, Y 62.7078, Z -6.3333, A 0.000, B 0.000, C 0.000 }
gfCNCPoint4[29542] = {X 273.8474, Y 62.2442, Z -6.3333, A 0.000, B 0.000, C 0.000 }
gfCNCPoint4[29543] = {X 273.1435, Y 61.5992, Z -6.3333, A 0.000, B 0.000, C 0.000 }
gfCNCPoint4[29544] = {X 272.6087, Y 60.8084, Z -6.3333, A 0.000, B 0.000, C 0.000 }
gfCNCPoint4[29545] = {X 272.2723, Y 59.9149, Z -6.3333, A 0.000, B 0.000, C 0.000 }
gfCNCPoint4[29546] = {X 272.1528, Y 58.9678, Z -6.3333, A 0.000, B 0.000, C 0.000 }
gfCNCPoint4[29547] = {X 272.1527, Y 58.0000, Z -6.3333, A 0.000, B 0.000, C 0.000 }
gfCNCPoint4[29548] = {X 272.2550, Y 57.0921, Z -6.3333, A 0.000, B 0.000, C 0.000 }
gfCNCPoint4[29549] = {X 272.5567, Y 56.2298, Z -6.3333, A 0.000, B 0.000, C 0.000 }
gfCNCPoint4[29550] = {X 273.0428, Y 55.4562, Z -6.3333, A 0.000, B 0.000, C 0.000 }
gfCNCPoint4[29551] = {X 273.6889, Y 54.8101, Z -6.3333, A 0.000, B 0.000, C 0.000 }
gfCNCPoint4[29552] = {X 274.4624, Y 54.3240, Z -6.3333, A 0.000, B 0.000, C 0.000 }
gfCNCPoint4[29553] = {X 275.3248, Y 54.0223, Z -6.3333, A 0.000, B 0.000, C 0.000 }
gfCNCPoint4[29554] = {X 276.2327, Y 53.9200, Z -6.3333, A 0.000, B 0.000, C 0.000 }
gfCNCPoint4[29555] = {X 292.7731, Y 53.9200, Z -6.3333, A 0.000, B 0.000, C 0.000 }
gfCNCPoint4[29556] = {X 293.6810, Y 54.0223, Z -6.3333, A 0.000, B 0.000, C 0.000 }
gfCNCPoint4[29557] = {X 294.5433, Y 54.3240, Z -6.3333, A 0.000, B 0.000, C 0.000 }
gfCNCPoint4[29558] = {X 295.3169, Y 54.8101, Z -6.3333, A 0.000, B 0.000, C 0.000 }
gfCNCPoint4[29559] = {X 295.9630, Y 55.4562, Z -6.3333, A 0.000, B 0.000, C 0.000 }
gfCNCPoint4[29560] = {X 296.4490, Y 56.2298, Z -6.3333, A 0.000, B 0.000, C 0.000 }
gfCNCPoint4[29561] = {X 296.7508, Y 57.0921, Z -6.3333, A 0.000, B 0.000, C 0.000 }
gfCNCPoint4[29562] = {X 296.8531, Y 58.0000, Z -6.3333, A 0.000, B 0.000, C 0.000 }
gfCNCPoint4[29563] = {X 296.8531, Y 58.9343, Z -6.3333, A 0.000, B 0.000, C 0.000 }
gfCNCPoint4[29564] = {X 296.7378, Y 59.8875, Z -6.3333, A 0.000, B 0.000, C 0.000 }
gfCNCPoint4[29565] = {X 296.4039, Y 60.7876, Z -6.3333, A 0.000, B 0.000, C 0.000 }
gfCNCPoint4[29566] = {X 295.8696, Y 61.5853, Z -6.3333, A 0.000, B 0.000, C 0.000 }
gfCNCPoint4[29567] = {X 295.1643, Y 62.2366, Z -6.3333, A 0.000, B 0.000, C 0.000 }
gfCNCPoint4[29568] = {X 294.3267, Y 62.7060, Z -6.3333, A 0.000, B 0.000, C 0.000 }
gfCNCPoint4[29569] = {X 293.4030, Y 62.9675, Z -6.3333, A 0.000, B 0.000, C 0.000 }
gfCNCPoint4[29570] = {X 293.2760, Y 62.9857, Z -6.3333, A 0.000, B 0.000, C 0.000 }
gfCNCPoint4[29571] = {X 293.1485, Y 63.0000, Z -6.3333, A 0.000, B 0.000, C 0.000 }
gfCNCPoint4[29572] = {X 293.1334, Y 63.1578, Z -6.3333, A 0.000, B 0.000, C 0.000 }
gfCNCPoint4[29573] = {X 293.1448, Y 92.9925, Z -6.3333, A 0.000, B 0.000, C 0.000 }
gfCNCPoint4[29574] = {X 293.2737, Y 93.0072, Z -6.3333, A 0.000, B 0.000, C 0.000 }
gfCNCPoint4[29575] = {X 293.4020, Y 93.0261, Z -6.3333, A 0.000, B 0.000, C 0.000 }
gfCNCPoint4[29576] = {X 294.3255, Y 93.2902, Z -6.3333, A 0.000, B 0.000, C 0.000 }
gfCNCPoint4[29577] = {X 295.1625, Y 93.7613, Z -6.3333, A 0.000, B 0.000, C 0.000 }
gfCNCPoint4[29578] = {X 295.8674, Y 94.4138, Z -6.3333, A 0.000, B 0.000, C 0.000 }
gfCNCPoint4[29579] = {X 296.4018, Y 95.2119, Z -6.3333, A 0.000, B 0.000, C 0.000 }
gfCNCPoint4[29580] = {X 296.7364, Y 96.1123, Z -6.3333, A 0.000, B 0.000, C 0.000 }
gfCNCPoint4[29581] = {X 296.8531, Y 97.0657, Z -6.3333, A 0.000, B 0.000, C 0.000 }
gfCNCPoint4[29582] = {X 296.8531, Y 98.0000, Z -6.3333, A 0.000, B 0.000, C 0.000 }
gfCNCPoint4[29583] = {X 296.7508, Y 98.9079, Z -6.3333, A 0.000, B 0.000, C 0.000 }
gfCNCPoint4[29584] = {X 296.4490, Y 99.7702, Z -6.3333, A 0.000, B 0.000, C 0.000 }
gfCNCPoint4[29585] = {X 295.9630, Y 100.5438, Z -6.3333, A 0.000, B 0.000, C 0.000 }
gfCNCPoint4[29586] = {X 295.3169, Y 101.1899, Z -6.3333, A 0.000, B 0.000, C 0.000 }
gfCNCPoint4[29587] = {X 294.5433, Y 101.6760, Z -6.3333, A 0.000, B 0.000, C 0.000 }
gfCNCPoint4[29588] = {X 293.6810, Y 101.9777, Z -6.3333, A 0.000, B 0.000, C 0.000 }
gfCNCPoint4[29589] = {X 292.7731, Y 102.0800, Z -6.3333, A 0.000, B 0.000, C 0.000 }
gfCNCPoint4[29590] = {X 276.2327, Y 102.0800, Z -6.3333, A 0.000, B 0.000, C 0.000 }
gfCNCPoint4[29591] = {X 275.3248, Y 101.9777, Z -6.3333, A 0.000, B 0.000, C 0.000 }
gfCNCPoint4[29592] = {X 274.4624, Y 101.6760, Z -6.3333, A 0.000, B 0.000, C 0.000 }
gfCNCPoint4[29593] = {X 273.6889, Y 101.1899, Z -6.3333, A 0.000, B 0.000, C 0.000 }
gfCNCPoint4[29594] = {X 273.0428, Y 100.5438, Z -6.3333, A 0.000, B 0.000, C 0.000 }
gfCNCPoint4[29595] = {X 272.5567, Y 99.7702, Z -6.3333, A 0.000, B 0.000, C 0.000 }
gfCNCPoint4[29596] = {X 272.2550, Y 98.9079, Z -6.3333, A 0.000, B 0.000, C 0.000 }
gfCNCPoint4[29597] = {X 272.1527, Y 98.0000, Z -6.3333, A 0.000, B 0.000, C 0.000 }
gfCNCPoint4[29598] = {X 272.1527, Y 97.0659, Z -6.3333, A 0.000, B 0.000, C 0.000 }
gfCNCPoint4[29599] = {X 272.2438, Y 96.2087, Z -6.3333, A 0.000, B 0.000, C 0.000 }
gfCNCPoint4[29600] = {X 272.5129, Y 95.3898, Z -6.3333, A 0.000, B 0.000, C 0.000 }
gfCNCPoint4[29601] = {X 272.9480, Y 94.6458, Z -6.3333, A 0.000, B 0.000, C 0.000 }
gfCNCPoint4[29602] = {X 273.5297, Y 94.0097, Z -6.3333, A 0.000, B 0.000, C 0.000 }
gfCNCPoint4[29603] = {X 274.2321, Y 93.5101, Z -6.3333, A 0.000, B 0.000, C 0.000 }
gfCNCPoint4[29604] = {X 275.0238, Y 93.1692, Z -6.3333, A 0.000, B 0.000, C 0.000 }
gfCNCPoint4[29605] = {X 275.8694, Y 93.0021, Z -6.3333, A 0.000, B 0.000, C 0.000 }
gfCNCPoint4[29606] = {X 275.8694, Y 85.4313, Z -6.3333, A 0.000, B 0.000, C 0.000 }
gfCNCPoint4[29607] = {X 262.6143, Y 80.2353, Z -6.3333, A 0.000, B 0.000, C 0.000 }
gfCNCPoint4[29608] = {X 262.1485, Y 80.5294, Z -6.3333, A 0.000, B 0.000, C 0.000 }
gfCNCPoint4[29609] = {X 237.5564, Y 96.4583, Z -6.3333, A 0.000, B 0.000, C 0.000 }
gfCNCPoint4[29610] = {X 237.5598, Y 97.0657, Z -6.3333, A 0.000, B 0.000, C 0.000 }
gfCNCPoint4[29611] = {X 237.5598, Y 98.0000, Z -6.3333, A 0.000, B 0.000, C 0.000 }
gfCNCPoint4[29612] = {X 237.4575, Y 98.9079, Z -6.3333, A 0.000, B 0.000, C 0.000 }
gfCNCPoint4[29613] = {X 237.1557, Y 99.7702, Z -6.3333, A 0.000, B 0.000, C 0.000 }
gfCNCPoint4[29614] = {X 236.6697, Y 100.5438, Z -6.3333, A 0.000, B 0.000, C 0.000 }
gfCNCPoint4[29615] = {X 236.0236, Y 101.1899, Z -6.3333, A 0.000, B 0.000, C 0.000 }
gfCNCPoint4[29616] = {X 235.2500, Y 101.6760, Z -6.3333, A 0.000, B 0.000, C 0.000 }
gfCNCPoint4[29617] = {X 234.3877, Y 101.9777, Z -6.3333, A 0.000, B 0.000, C 0.000 }
gfCNCPoint4[29618] = {X 233.4798, Y 102.0800, Z -6.3333, A 0.000, B 0.000, C 0.000 }
gfCNCPoint4[29619] = {X 214.1790, Y 102.0800, Z -6.3333, A 0.000, B 0.000, C 0.000 }
gfCNCPoint4[29620] = {X 213.7860, Y 102.0610, Z -6.3333, A 0.000, B 0.000, C 0.000 }
gfCNCPoint4[29621] = {X 213.3966, Y 102.0043, Z -6.3333, A 0.000, B 0.000, C 0.000 }
gfCNCPoint4[29622] = {X 213.0072, Y 102.0610, Z -6.3333, A 0.000, B 0.000, C 0.000 }
gfCNCPoint4[29623] = {X 212.6141, Y 102.0800, Z -6.3333, A 0.000, B 0.000, C 0.000 }
gfCNCPoint4[29624] = {X 194.9870, Y 102.0800, Z -6.3333, A 0.000, B 0.000, C 0.000 }
gfCNCPoint4[29625] = {X 194.0791, Y 101.9777, Z -6.3333, A 0.000, B 0.000, C 0.000 }
gfCNCPoint4[29626] = {X 193.2167, Y 101.6760, Z -6.3333, A 0.000, B 0.000, C 0.000 }
gfCNCPoint4[29627] = {X 192.4431, Y 101.1899, Z -6.3333, A 0.000, B 0.000, C 0.000 }
gfCNCPoint4[29628] = {X 191.7971, Y 100.5438, Z -6.3333, A 0.000, B 0.000, C 0.000 }
gfCNCPoint4[29629] = {X 191.3110, Y 99.7702, Z -6.3333, A 0.000, B 0.000, C 0.000 }
gfCNCPoint4[29630] = {X 191.0093, Y 98.9079, Z -6.3333, A 0.000, B 0.000, C 0.000 }
gfCNCPoint4[29631] = {X 190.9070, Y 98.0000, Z -6.3333, A 0.000, B 0.000, C 0.000 }
gfCNCPoint4[29632] = {X 190.9070, Y 97.0659, Z -6.3333, A 0.000, B 0.000, C 0.000 }
gfCNCPoint4[29633] = {X 191.0022, Y 96.1894, Z -6.3333, A 0.000, B 0.000, C 0.000 }
gfCNCPoint4[29634] = {X 191.2835, Y 95.3539, Z -6.3333, A 0.000, B 0.000, C 0.000 }
gfCNCPoint4[29635] = {X 191.7378, Y 94.5983, Z -6.3333, A 0.000, B 0.000, C 0.000 }
gfCNCPoint4[29636] = {X 191.8199, Y 94.4938, Z -6.3333, A 0.000, B 0.000, C 0.000 }
gfCNCPoint4[29637] = {X 191.9053, Y 94.3920, Z -6.3333, A 0.000, B 0.000, C 0.000 }
gfCNCPoint4[29638] = {X 188.6703, Y 90.8602, Z -6.3333, A 0.000, B 0.000, C 0.000 }
gfCNCPoint4[29639] = {X 149.9831, Y 90.8602, Z -6.3333, A 0.000, B 0.000, C 0.000 }
gfCNCPoint4[29640] = {X 146.8270, Y 94.3569, Z -6.3333, A 0.000, B 0.000, C 0.000 }
gfCNCPoint4[29641] = {X 147.3874, Y 95.1673, Z -6.3333, A 0.000, B 0.000, C 0.000 }
gfCNCPoint4[29642] = {X 147.7382, Y 96.0880, Z -6.3333, A 0.000, B 0.000, C 0.000 }
gfCNCPoint4[29643] = {X 147.8591, Y 97.0659, Z -6.3333, A 0.000, B 0.000, C 0.000 }
gfCNCPoint4[29644] = {X 147.8591, Y 98.0000, Z -6.3333, A 0.000, B 0.000, C 0.000 }
gfCNCPoint4[29645] = {X 147.7568, Y 98.9079, Z -6.3333, A 0.000, B 0.000, C 0.000 }
gfCNCPoint4[29646] = {X 147.4551, Y 99.7702, Z -6.3333, A 0.000, B 0.000, C 0.000 }
gfCNCPoint4[29647] = {X 146.9690, Y 100.5438, Z -6.3333, A 0.000, B 0.000, C 0.000 }
gfCNCPoint4[29648] = {X 146.3229, Y 101.1899, Z -6.3333, A 0.000, B 0.000, C 0.000 }
gfCNCPoint4[29649] = {X 145.5494, Y 101.6760, Z -6.3333, A 0.000, B 0.000, C 0.000 }
gfCNCPoint4[29650] = {X 144.6870, Y 101.9777, Z -6.3333, A 0.000, B 0.000, C 0.000 }
gfCNCPoint4[29651] = {X 143.7791, Y 102.0800, Z -6.3333, A 0.000, B 0.000, C 0.000 }
gfCNCPoint4[29652] = {X 125.0000, Y 102.0800, Z -6.3333, A 0.000, B 0.000, C 0.000 }
gfCNCPoint4[29653] = {X 124.0921, Y 101.9777, Z -6.3333, A 0.000, B 0.000, C 0.000 }
gfCNCPoint4[29654] = {X 123.2298, Y 101.6760, Z -6.3333, A 0.000, B 0.000, C 0.000 }
gfCNCPoint4[29655] = {X 122.4562, Y 101.1899, Z -6.3333, A 0.000, B 0.000, C 0.000 }
gfCNCPoint4[29656] = {X 121.8101, Y 100.5438, Z -6.3333, A 0.000, B 0.000, C 0.000 }
gfCNCPoint4[29657] = {X 121.3240, Y 99.7702, Z -6.3333, A 0.000, B 0.000, C 0.000 }
gfCNCPoint4[29658] = {X 121.0223, Y 98.9079, Z -6.3333, A 0.000, B 0.000, C 0.000 }
gfCNCPoint4[29659] = {X 120.9200, Y 98.0000, Z -6.3333, A 0.000, B 0.000, C 0.000 }
gfCNCPoint4[29660] = {X 120.9200, Y 97.0659, Z -6.3333, A 0.000, B 0.000, C 0.000 }
gfCNCPoint4[29661] = {X 121.0193, Y 96.1711, Z -6.3333, A 0.000, B 0.000, C 0.000 }
gfCNCPoint4[29662] = {X 121.3125, Y 95.3198, Z -6.3333, A 0.000, B 0.000, C 0.000 }
gfCNCPoint4[29663] = {X 121.7853, Y 94.5535, Z -6.3333, A 0.000, B 0.000, C 0.000 }
gfCNCPoint4[29664] = {X 122.4147, Y 93.9096, Z -6.3333, A 0.000, B 0.000, C 0.000 }
gfCNCPoint4[29665] = {X 123.1699, Y 93.4194, Z -6.3333, A 0.000, B 0.000, C 0.000 }
gfCNCPoint4[29666] = {X 124.0143, Y 93.1068, Z -6.3333, A 0.000, B 0.000, C 0.000 }
gfCNCPoint4[29667] = {X 124.9066, Y 92.9870, Z -6.3333, A 0.000, B 0.000, C 0.000 }
gfCNCPoint4[29668] = {X 124.9295, Y 92.9713, Z -6.3333, A 0.000, B 0.000, C 0.000 }
gfCNCPoint4[29669] = {X 124.9630, Y 92.9582, Z -6.3333, A 0.000, B 0.000, C 0.000 }
gfCNCPoint4[29670] = {X 125.4829, Y 92.8811, Z -6.3333, A 0.000, B 0.000, C 0.000 }
gfCNCPoint4[29671] = {X 126.3567, Y 92.7330, Z -6.3333, A 0.000, B 0.000, C 0.000 }
gfCNCPoint4[29672] = {X 127.2179, Y 92.5235, Z -6.3333, A 0.000, B 0.000, C 0.000 }
gfCNCPoint4[29673] = {X 128.4708, Y 91.3460, Z -6.3333, A 0.000, B 0.000, C 0.000 }
gfCNCPoint4[29674] = {X 129.6565, Y 90.1009, Z -6.3333, A 0.000, B 0.000, C 0.000 }
gfCNCPoint4[29675] = {X 140.8574, Y 77.8008, Z -6.3333, A 0.000, B 0.000, C 0.000 }
gfCNCPoint4[29676] = {X 137.9000, Y 75.1076, Z -6.3333, A 0.000, B 0.000, C 0.000 }
gfCNCPoint4[29677] = {X 140.9166, Y 77.8546, Z -6.3333, A 0.000, B 0.000, C 0.000 }
gfCNCPoint4[29678] = {X 156.0369, Y 61.2504, Z -6.3333, A 0.000, B 0.000, C 0.000 }
gfCNCPoint4[29679] = {X 155.6323, Y 60.5349, Z -6.3333, A 0.000, B 0.000, C 0.000 }
gfCNCPoint4[29680] = {X 155.3824, Y 59.7517, Z -6.3333, A 0.000, B 0.000, C 0.000 }
gfCNCPoint4[29681] = {X 155.2980, Y 58.9341, Z -6.3333, A 0.000, B 0.000, C 0.000 }
gfCNCPoint4[29682] = {X 155.2980, Y 58.0000, Z -6.3333, A 0.000, B 0.000, C 0.000 }
gfCNCPoint4[29683] = {X 155.3982, Y 57.1099, Z -6.3333, A 0.000, B 0.000, C 0.000 }
gfCNCPoint4[29684] = {X 155.6941, Y 56.2645, Z -6.3333, A 0.000, B 0.000, C 0.000 }
gfCNCPoint4[29685] = {X 156.1706, Y 55.5060, Z -6.3333, A 0.000, B 0.000, C 0.000 }
gfCNCPoint4[29686] = {X 156.8040, Y 54.8727, Z -6.3333, A 0.000, B 0.000, C 0.000 }
gfCNCPoint4[29687] = {X 157.5624, Y 54.3961, Z -6.3333, A 0.000, B 0.000, C 0.000 }
gfCNCPoint4[29688] = {X 158.4079, Y 54.1003, Z -6.3333, A 0.000, B 0.000, C 0.000 }
gfCNCPoint4[29689] = {X 159.2980, Y 54.0000, Z -6.3333, A 0.000, B 0.000, C 0.000 }
gfCNCPoint4[29690] = {X 178.5335, Y 54.0000, Z -6.3333, A 0.000, B 0.000, C 0.000 }
gfCNCPoint4[29691] = {X 179.4236, Y 54.1003, Z -6.3333, A 0.000, B 0.000, C 0.000 }
gfCNCPoint4[29692] = {X 180.2690, Y 54.3961, Z -6.3333, A 0.000, B 0.000, C 0.000 }
gfCNCPoint4[29693] = {X 181.0275, Y 54.8727, Z -6.3333, A 0.000, B 0.000, C 0.000 }
gfCNCPoint4[29694] = {X 181.6608, Y 55.5060, Z -6.3333, A 0.000, B 0.000, C 0.000 }
gfCNCPoint4[29695] = {X 182.1374, Y 56.2645, Z -6.3333, A 0.000, B 0.000, C 0.000 }
gfCNCPoint4[29696] = {X 182.4332, Y 57.1099, Z -6.3333, A 0.000, B 0.000, C 0.000 }
gfCNCPoint4[29697] = {X 182.5335, Y 58.0000, Z -6.3333, A 0.000, B 0.000, C 0.000 }
gfCNCPoint4[29698] = {X 182.5334, Y 58.9671, Z -6.3333, A 0.000, B 0.000, C 0.000 }
gfCNCPoint4[29699] = {X 182.4464, Y 59.7645, Z -6.3333, A 0.000, B 0.000, C 0.000 }
gfCNCPoint4[29700] = {X 182.2020, Y 60.5284, Z -6.3333, A 0.000, B 0.000, C 0.000 }
gfCNCPoint4[29701] = {X 181.8102, Y 61.2283, Z -6.3333, A 0.000, B 0.000, C 0.000 }
gfCNCPoint4[29702] = {X 209.2437, Y 91.1705, Z -6.3333, A 0.000, B 0.000, C 0.000 }
gfCNCPoint4[29703] = {X 209.9165, Y 91.8531, Z -6.3333, A 0.000, B 0.000, C 0.000 }
gfCNCPoint4[29704] = {X 210.6372, Y 92.4850, Z -6.3333, A 0.000, B 0.000, C 0.000 }
gfCNCPoint4[29705] = {X 210.9789, Y 92.7008, Z -6.3333, A 0.000, B 0.000, C 0.000 }
gfCNCPoint4[29706] = {X 211.3621, Y 92.8291, Z -6.3333, A 0.000, B 0.000, C 0.000 }
gfCNCPoint4[29707] = {X 212.0545, Y 92.9772, Z -6.3333, A 0.000, B 0.000, C 0.000 }
gfCNCPoint4[29708] = {X 213.3961, Y 93.1462, Z -6.3333, A 0.000, B 0.000, C 0.000 }
gfCNCPoint4[29709] = {X 214.4555, Y 93.0559, Z -6.3333, A 0.000, B 0.000, C 0.000 }
gfCNCPoint4[29710] = {X 215.5170, Y 92.9948, Z -6.3333, A 0.000, B 0.000, C 0.000 }
gfCNCPoint4[29711] = {X 216.2444, Y 92.9147, Z -6.3333, A 0.000, B 0.000, C 0.000 }
gfCNCPoint4[29712] = {X 216.9448, Y 92.7025, Z -6.3333, A 0.000, B 0.000, C 0.000 }
gfCNCPoint4[29713] = {X 217.5944, Y 92.3653, Z -6.3333, A 0.000, B 0.000, C 0.000 }
gfCNCPoint4[29714] = {X 223.1343, Y 88.7902, Z -6.3333, A 0.000, B 0.000, C 0.000 }
gfCNCPoint4[29715] = {X 246.5287, Y 73.8311, Z -6.3333, A 0.000, B 0.000, C 0.000 }
gfCNCPoint4[29716] = {X 221.7493, Y 64.1072, Z -6.3333, A 0.000, B 0.000, C 0.000 }
gfCNCPoint4[29717] = {X 219.9471, Y 63.5041, Z -6.3333, A 0.000, B 0.000, C 0.000 }
gfCNCPoint4[29718] = {X 218.0878, Y 63.1105, Z -6.3333, A 0.000, B 0.000, C 0.000 }
gfCNCPoint4[29719] = {X 216.1958, Y 62.9318, Z -6.3333, A 0.000, B 0.000, C 0.000 }
gfCNCPoint4[29720] = {X 215.3283, Y 62.8064, Z -6.3333, A 0.000, B 0.000, C 0.000 }
gfCNCPoint4[29721] = {X 214.5089, Y 62.4951, Z -6.3333, A 0.000, B 0.000, C 0.000 }
gfCNCPoint4[29722] = {X 213.7770, Y 62.0127, Z -6.3333, A 0.000, B 0.000, C 0.000 }
gfCNCPoint4[29723] = {X 213.1677, Y 61.3825, Z -6.3333, A 0.000, B 0.000, C 0.000 }
gfCNCPoint4[29724] = {X 212.7104, Y 60.6348, Z -6.3333, A 0.000, B 0.000, C 0.000 }
gfCNCPoint4[29725] = {X 212.4268, Y 59.8053, Z -6.3333, A 0.000, B 0.000, C 0.000 }
gfCNCPoint4[29726] = {X 212.3308, Y 58.9341, Z -6.3333, A 0.000, B 0.000, C 0.000 }
gfCNCPoint4[29727] = {X 212.3308, Y 58.0000, Z -6.3333, A 0.000, B 0.000, C 0.000 }
gfCNCPoint4[29728] = {X 212.4311, Y 57.1099, Z -6.3333, A 0.000, B 0.000, C 0.000 }
gfCNCPoint4[29729] = {X 212.7269, Y 56.2645, Z -6.3333, A 0.000, B 0.000, C 0.000 }
gfCNCPoint4[29730] = {X 213.2035, Y 55.5060, Z -6.3333, A 0.000, B 0.000, C 0.000 }
gfCNCPoint4[29731] = {X 213.8368, Y 54.8727, Z -6.3333, A 0.000, B 0.000, C 0.000 }
gfCNCPoint4[29732] = {X 214.5953, Y 54.3961, Z -6.3333, A 0.000, B 0.000, C 0.000 }
gfCNCPoint4[29733] = {X 215.4407, Y 54.1003, Z -6.3333, A 0.000, B 0.000, C 0.000 }
gfCNCPoint4[29734] = {X 216.3308, Y 54.0000, Z -6.3333, A 0.000, B 0.000, C 0.000 }
gfCNCPoint4[29735] = {X 237.2617, Y 54.0000, Z -6.3333, A 0.000, B 0.000, C 0.000 }
gfCNCPoint4[29736] = {X 238.1518, Y 54.1003, Z -6.3333, A 0.000, B 0.000, C 0.000 }
gfCNCPoint4[29737] = {X 238.9972, Y 54.3961, Z -6.3333, A 0.000, B 0.000, C 0.000 }
gfCNCPoint4[29738] = {X 239.7556, Y 54.8727, Z -6.3333, A 0.000, B 0.000, C 0.000 }
gfCNCPoint4[29739] = {X 240.3890, Y 55.5060, Z -6.3333, A 0.000, B 0.000, C 0.000 }
gfCNCPoint4[29740] = {X 240.8656, Y 56.2645, Z -6.3333, A 0.000, B 0.000, C 0.000 }
gfCNCPoint4[29741] = {X 241.1614, Y 57.1099, Z -6.3333, A 0.000, B 0.000, C 0.000 }
gfCNCPoint4[29742] = {X 241.2617, Y 58.0000, Z -6.3333, A 0.000, B 0.000, C 0.000 }
gfCNCPoint4[29743] = {X 241.2617, Y 58.4506, Z -6.3333, A 0.000, B 0.000, C 0.000 }
gfCNCPoint4[29744] = {X 247.9973, Y 61.0771, Z -6.3333, A 0.000, B 0.000, C 0.000 }
gfCNCPoint4[29745] = {X 275.9522, Y 72.1729, Z -6.3333, A 0.000, B 0.000, C 0.000 }
gfCNCPoint4[29746] = {X 275.9518, Y 63.0392, Z -6.3333, A 0.000, B 0.000, C 0.000 }
gfCNCPoint4[29747] = {X 275.9573, Y 62.9246, Z -6.3333, A 0.000, B 0.000, C 0.000 }
gfCNCPoint4[29748] = {X 275.7851, Y 62.9089, Z -6.3333, A 0.000, B 0.000, C 0.000 }
gfCNCPoint4[29749] = {X 275.6137, Y 62.8859, Z -6.3333, A 0.000, B 0.000, C 0.000 }
gfCNCPoint4[29750] = {X 274.7072, Y 62.6318, Z -6.3333, A 0.000, B 0.000, C 0.000 }
gfCNCPoint4[29751] = {X 273.8852, Y 62.1728, Z -6.3333, A 0.000, B 0.000, C 0.000 }
gfCNCPoint4[29752] = {X 273.1933, Y 61.5344, Z -6.3333, A 0.000, B 0.000, C 0.000 }
gfCNCPoint4[29753] = {X 272.6697, Y 60.7520, Z -6.3333, A 0.000, B 0.000, C 0.000 }
gfCNCPoint4[29754] = {X 272.3435, Y 59.8689, Z -6.3333, A 0.000, B 0.000, C 0.000 }
gfCNCPoint4[29755] = {X 272.2327, Y 58.9341, Z -6.3333, A 0.000, B 0.000, C 0.000 }
gfCNCPoint4[29756] = {X 272.2327, Y 58.0000, Z -6.3333, A 0.000, B 0.000, C 0.000 }
gfCNCPoint4[29757] = {X 272.3330, Y 57.1099, Z -6.3333, A 0.000, B 0.000, C 0.000 }
gfCNCPoint4[29758] = {X 272.6288, Y 56.2645, Z -6.3333, A 0.000, B 0.000, C 0.000 }
gfCNCPoint4[29759] = {X 273.1054, Y 55.5060, Z -6.3333, A 0.000, B 0.000, C 0.000 }
gfCNCPoint4[29760] = {X 273.7387, Y 54.8727, Z -6.3333, A 0.000, B 0.000, C 0.000 }
gfCNCPoint4[29761] = {X 274.4972, Y 54.3961, Z -6.3333, A 0.000, B 0.000, C 0.000 }
gfCNCPoint4[29762] = {X 275.3426, Y 54.1003, Z -6.3333, A 0.000, B 0.000, C 0.000 }
gfCNCPoint4[29763] = {X 276.2327, Y 54.0000, Z -6.3333, A 0.000, B 0.000, C 0.000 }
gfCNCPoint4[29764] = {X 292.7731, Y 54.0000, Z -6.3333, A 0.000, B 0.000, C 0.000 }
gfCNCPoint4[29765] = {X 293.6632, Y 54.1003, Z -6.3333, A 0.000, B 0.000, C 0.000 }
gfCNCPoint4[29766] = {X 294.5086, Y 54.3961, Z -6.3333, A 0.000, B 0.000, C 0.000 }
gfCNCPoint4[29767] = {X 295.2670, Y 54.8727, Z -6.3333, A 0.000, B 0.000, C 0.000 }
gfCNCPoint4[29768] = {X 295.9004, Y 55.5060, Z -6.3333, A 0.000, B 0.000, C 0.000 }
gfCNCPoint4[29769] = {X 296.3770, Y 56.2645, Z -6.3333, A 0.000, B 0.000, C 0.000 }
gfCNCPoint4[29770] = {X 296.6728, Y 57.1099, Z -6.3333, A 0.000, B 0.000, C 0.000 }
gfCNCPoint4[29771] = {X 296.7731, Y 58.0000, Z -6.3333, A 0.000, B 0.000, C 0.000 }
gfCNCPoint4[29772] = {X 296.7731, Y 58.9341, Z -6.3333, A 0.000, B 0.000, C 0.000 }
gfCNCPoint4[29773] = {X 296.6601, Y 59.8686, Z -6.3333, A 0.000, B 0.000, C 0.000 }
gfCNCPoint4[29774] = {X 296.3326, Y 60.7512, Z -6.3333, A 0.000, B 0.000, C 0.000 }
gfCNCPoint4[29775] = {X 295.8088, Y 61.5333, Z -6.3333, A 0.000, B 0.000, C 0.000 }
gfCNCPoint4[29776] = {X 295.1173, Y 62.1719, Z -6.3333, A 0.000, B 0.000, C 0.000 }
gfCNCPoint4[29777] = {X 294.2961, Y 62.6321, Z -6.3333, A 0.000, B 0.000, C 0.000 }
gfCNCPoint4[29778] = {X 293.3903, Y 62.8885, Z -6.3333, A 0.000, B 0.000, C 0.000 }
gfCNCPoint4[29779] = {X 293.2331, Y 62.9104, Z -6.3333, A 0.000, B 0.000, C 0.000 }
gfCNCPoint4[29780] = {X 293.0752, Y 62.9261, Z -6.3333, A 0.000, B 0.000, C 0.000 }
gfCNCPoint4[29781] = {X 293.0534, Y 63.1540, Z -6.3333, A 0.000, B 0.000, C 0.000 }
gfCNCPoint4[29782] = {X 293.0534, Y 92.9237, Z -6.3333, A 0.000, B 0.000, C 0.000 }
gfCNCPoint4[29783] = {X 293.0752, Y 93.0665, Z -6.3333, A 0.000, B 0.000, C 0.000 }
gfCNCPoint4[29784] = {X 293.2325, Y 93.0827, Z -6.3333, A 0.000, B 0.000, C 0.000 }
gfCNCPoint4[29785] = {X 293.3891, Y 93.1050, Z -6.3333, A 0.000, B 0.000, C 0.000 }
gfCNCPoint4[29786] = {X 294.2946, Y 93.3640, Z -6.3333, A 0.000, B 0.000, C 0.000 }
gfCNCPoint4[29787] = {X 295.1154, Y 93.8260, Z -6.3333, A 0.000, B 0.000, C 0.000 }
gfCNCPoint4[29788] = {X 295.8066, Y 94.4657, Z -6.3333, A 0.000, B 0.000, C 0.000 }
gfCNCPoint4[29789] = {X 296.3306, Y 95.2484, Z -6.3333, A 0.000, B 0.000, C 0.000 }
gfCNCPoint4[29790] = {X 296.6587, Y 96.1312, Z -6.3333, A 0.000, B 0.000, C 0.000 }
gfCNCPoint4[29791] = {X 296.7731, Y 97.0660, Z -6.3333, A 0.000, B 0.000, C 0.000 }
gfCNCPoint4[29792] = {X 296.7731, Y 98.0000, Z -6.3333, A 0.000, B 0.000, C 0.000 }
gfCNCPoint4[29793] = {X 296.6728, Y 98.8901, Z -6.3333, A 0.000, B 0.000, C 0.000 }
gfCNCPoint4[29794] = {X 296.3770, Y 99.7355, Z -6.3333, A 0.000, B 0.000, C 0.000 }
gfCNCPoint4[29795] = {X 295.9004, Y 100.4940, Z -6.3333, A 0.000, B 0.000, C 0.000 }
gfCNCPoint4[29796] = {X 295.2670, Y 101.1273, Z -6.3333, A 0.000, B 0.000, C 0.000 }
gfCNCPoint4[29797] = {X 294.5086, Y 101.6039, Z -6.3333, A 0.000, B 0.000, C 0.000 }
gfCNCPoint4[29798] = {X 293.6632, Y 101.8997, Z -6.3333, A 0.000, B 0.000, C 0.000 }
gfCNCPoint4[29799] = {X 292.7731, Y 102.0000, Z -6.3333, A 0.000, B 0.000, C 0.000 }
gfCNCPoint4[29800] = {X 276.2327, Y 102.0000, Z -6.3333, A 0.000, B 0.000, C 0.000 }
gfCNCPoint4[29801] = {X 275.3426, Y 101.8997, Z -6.3333, A 0.000, B 0.000, C 0.000 }
gfCNCPoint4[29802] = {X 274.4972, Y 101.6039, Z -6.3333, A 0.000, B 0.000, C 0.000 }
gfCNCPoint4[29803] = {X 273.7387, Y 101.1273, Z -6.3333, A 0.000, B 0.000, C 0.000 }
gfCNCPoint4[29804] = {X 273.1054, Y 100.4940, Z -6.3333, A 0.000, B 0.000, C 0.000 }
gfCNCPoint4[29805] = {X 272.6288, Y 99.7355, Z -6.3333, A 0.000, B 0.000, C 0.000 }
gfCNCPoint4[29806] = {X 272.3330, Y 98.8901, Z -6.3333, A 0.000, B 0.000, C 0.000 }
gfCNCPoint4[29807] = {X 272.2327, Y 98.0000, Z -6.3333, A 0.000, B 0.000, C 0.000 }
gfCNCPoint4[29808] = {X 272.2329, Y 97.0232, Z -6.3333, A 0.000, B 0.000, C 0.000 }
gfCNCPoint4[29809] = {X 272.3321, Y 96.1797, Z -6.3333, A 0.000, B 0.000, C 0.000 }
gfCNCPoint4[29810] = {X 272.6072, Y 95.3761, Z -6.3333, A 0.000, B 0.000, C 0.000 }
gfCNCPoint4[29811] = {X 273.0457, Y 94.6486, Z -6.3333, A 0.000, B 0.000, C 0.000 }
gfCNCPoint4[29812] = {X 273.6280, Y 94.0302, Z -6.3333, A 0.000, B 0.000, C 0.000 }
gfCNCPoint4[29813] = {X 274.3277, Y 93.5487, Z -6.3333, A 0.000, B 0.000, C 0.000 }
gfCNCPoint4[29814] = {X 275.1133, Y 93.2258, Z -6.3333, A 0.000, B 0.000, C 0.000 }
gfCNCPoint4[29815] = {X 275.9494, Y 93.0760, Z -6.3333, A 0.000, B 0.000, C 0.000 }
gfCNCPoint4[29816] = {X 275.9494, Y 85.3767, Z -6.3333, A 0.000, B 0.000, C 0.000 }
gfCNCPoint4[29817] = {X 262.6059, Y 80.1460, Z -6.3333, A 0.000, B 0.000, C 0.000 }
gfCNCPoint4[29818] = {X 262.1054, Y 80.4620, Z -6.3333, A 0.000, B 0.000, C 0.000 }
gfCNCPoint4[29819] = {X 237.4762, Y 96.4149, Z -6.3333, A 0.000, B 0.000, C 0.000 }
gfCNCPoint4[29820] = {X 237.4798, Y 97.0659, Z -6.3333, A 0.000, B 0.000, C 0.000 }
gfCNCPoint4[29821] = {X 237.4798, Y 98.0000, Z -6.3333, A 0.000, B 0.000, C 0.000 }
gfCNCPoint4[29822] = {X 237.3795, Y 98.8901, Z -6.3333, A 0.000, B 0.000, C 0.000 }
gfCNCPoint4[29823] = {X 237.0837, Y 99.7355, Z -6.3333, A 0.000, B 0.000, C 0.000 }
gfCNCPoint4[29824] = {X 236.6071, Y 100.4940, Z -6.3333, A 0.000, B 0.000, C 0.000 }
gfCNCPoint4[29825] = {X 235.9737, Y 101.1273, Z -6.3333, A 0.000, B 0.000, C 0.000 }
gfCNCPoint4[29826] = {X 235.2153, Y 101.6039, Z -6.3333, A 0.000, B 0.000, C 0.000 }
gfCNCPoint4[29827] = {X 234.3699, Y 101.8997, Z -6.3333, A 0.000, B 0.000, C 0.000 }
gfCNCPoint4[29828] = {X 233.4798, Y 102.0000, Z -6.3333, A 0.000, B 0.000, C 0.000 }
gfCNCPoint4[29829] = {X 214.1790, Y 102.0000, Z -6.3333, A 0.000, B 0.000, C 0.000 }
gfCNCPoint4[29830] = {X 213.7859, Y 101.9806, Z -6.3333, A 0.000, B 0.000, C 0.000 }
gfCNCPoint4[29831] = {X 213.3966, Y 101.9227, Z -6.3333, A 0.000, B 0.000, C 0.000 }
gfCNCPoint4[29832] = {X 213.0072, Y 101.9806, Z -6.3333, A 0.000, B 0.000, C 0.000 }
gfCNCPoint4[29833] = {X 212.6141, Y 102.0000, Z -6.3333, A 0.000, B 0.000, C 0.000 }
gfCNCPoint4[29834] = {X 194.9870, Y 102.0000, Z -6.3333, A 0.000, B 0.000, C 0.000 }
gfCNCPoint4[29835] = {X 194.0969, Y 101.8997, Z -6.3333, A 0.000, B 0.000, C 0.000 }
gfCNCPoint4[29836] = {X 193.2514, Y 101.6039, Z -6.3333, A 0.000, B 0.000, C 0.000 }
gfCNCPoint4[29837] = {X 192.4930, Y 101.1273, Z -6.3333, A 0.000, B 0.000, C 0.000 }
gfCNCPoint4[29838] = {X 191.8596, Y 100.4940, Z -6.3333, A 0.000, B 0.000, C 0.000 }
gfCNCPoint4[29839] = {X 191.3831, Y 99.7355, Z -6.3333, A 0.000, B 0.000, C 0.000 }
gfCNCPoint4[29840] = {X 191.0872, Y 98.8901, Z -6.3333, A 0.000, B 0.000, C 0.000 }
gfCNCPoint4[29841] = {X 190.9870, Y 98.0000, Z -6.3333, A 0.000, B 0.000, C 0.000 }
gfCNCPoint4[29842] = {X 190.9870, Y 97.0659, Z -6.3333, A 0.000, B 0.000, C 0.000 }
gfCNCPoint4[29843] = {X 191.0804, Y 96.2066, Z -6.3333, A 0.000, B 0.000, C 0.000 }
gfCNCPoint4[29844] = {X 191.3562, Y 95.3874, Z -6.3333, A 0.000, B 0.000, C 0.000 }
gfCNCPoint4[29845] = {X 191.8015, Y 94.6466, Z -6.3333, A 0.000, B 0.000, C 0.000 }
gfCNCPoint4[29846] = {X 191.9053, Y 94.5175, Z -6.3333, A 0.000, B 0.000, C 0.000 }
gfCNCPoint4[29847] = {X 192.0144, Y 94.3927, Z -6.3333, A 0.000, B 0.000, C 0.000 }
gfCNCPoint4[29848] = {X 188.7055, Y 90.7802, Z -6.3333, A 0.000, B 0.000, C 0.000 }
gfCNCPoint4[29849] = {X 149.9476, Y 90.7802, Z -6.3333, A 0.000, B 0.000, C 0.000 }
gfCNCPoint4[29850] = {X 146.7192, Y 94.3569, Z -6.3333, A 0.000, B 0.000, C 0.000 }
gfCNCPoint4[29851] = {X 147.1694, Y 94.9481, Z -6.3333, A 0.000, B 0.000, C 0.000 }
gfCNCPoint4[29852] = {X 147.5030, Y 95.6122, Z -6.3333, A 0.000, B 0.000, C 0.000 }
gfCNCPoint4[29853] = {X 147.7085, Y 96.3263, Z -6.3333, A 0.000, B 0.000, C 0.000 }
gfCNCPoint4[29854] = {X 147.7791, Y 97.0660, Z -6.3333, A 0.000, B 0.000, C 0.000 }
gfCNCPoint4[29855] = {X 147.7791, Y 98.0000, Z -6.3333, A 0.000, B 0.000, C 0.000 }
gfCNCPoint4[29856] = {X 147.6788, Y 98.8901, Z -6.3333, A 0.000, B 0.000, C 0.000 }
gfCNCPoint4[29857] = {X 147.3830, Y 99.7355, Z -6.3333, A 0.000, B 0.000, C 0.000 }
gfCNCPoint4[29858] = {X 146.9064, Y 100.4940, Z -6.3333, A 0.000, B 0.000, C 0.000 }
gfCNCPoint4[29859] = {X 146.2731, Y 101.1273, Z -6.3333, A 0.000, B 0.000, C 0.000 }
gfCNCPoint4[29860] = {X 145.5146, Y 101.6039, Z -6.3333, A 0.000, B 0.000, C 0.000 }
gfCNCPoint4[29861] = {X 144.6692, Y 101.8997, Z -6.3333, A 0.000, B 0.000, C 0.000 }
gfCNCPoint4[29862] = {X 143.7791, Y 102.0000, Z -6.3333, A 0.000, B 0.000, C 0.000 }
gfCNCPoint4[29863] = {X 125.0000, Y 102.0000, Z -6.3333, A 0.000, B 0.000, C 0.000 }
gfCNCPoint4[29864] = {X 124.1099, Y 101.8997, Z -6.3333, A 0.000, B 0.000, C 0.000 }
gfCNCPoint4[29865] = {X 123.2645, Y 101.6039, Z -6.3333, A 0.000, B 0.000, C 0.000 }
gfCNCPoint4[29866] = {X 122.5060, Y 101.1273, Z -6.3333, A 0.000, B 0.000, C 0.000 }
gfCNCPoint4[29867] = {X 121.8727, Y 100.4940, Z -6.3333, A 0.000, B 0.000, C 0.000 }
gfCNCPoint4[29868] = {X 121.3961, Y 99.7355, Z -6.3333, A 0.000, B 0.000, C 0.000 }
gfCNCPoint4[29869] = {X 121.1003, Y 98.8901, Z -6.3333, A 0.000, B 0.000, C 0.000 }
gfCNCPoint4[29870] = {X 121.0000, Y 98.0000, Z -6.3333, A 0.000, B 0.000, C 0.000 }
gfCNCPoint4[29871] = {X 121.0000, Y 97.0659, Z -6.3333, A 0.000, B 0.000, C 0.000 }
gfCNCPoint4[29872] = {X 121.0981, Y 96.1853, Z -6.3333, A 0.000, B 0.000, C 0.000 }
gfCNCPoint4[29873] = {X 121.3877, Y 95.3479, Z -6.3333, A 0.000, B 0.000, C 0.000 }
gfCNCPoint4[29874] = {X 121.8546, Y 94.5948, Z -6.3333, A 0.000, B 0.000, C 0.000 }
gfCNCPoint4[29875] = {X 122.4758, Y 93.9629, Z -6.3333, A 0.000, B 0.000, C 0.000 }
gfCNCPoint4[29876] = {X 123.2209, Y 93.4834, Z -6.3333, A 0.000, B 0.000, C 0.000 }
gfCNCPoint4[29877] = {X 124.0533, Y 93.1796, Z -6.3333, A 0.000, B 0.000, C 0.000 }
gfCNCPoint4[29878] = {X 124.9321, Y 93.0665, Z -6.3333, A 0.000, B 0.000, C 0.000 }
gfCNCPoint4[29879] = {X 124.9747, Y 93.0373, Z -6.3333, A 0.000, B 0.000, C 0.000 }
gfCNCPoint4[29880] = {X 125.4940, Y 92.9603, Z -6.3333, A 0.000, B 0.000, C 0.000 }
gfCNCPoint4[29881] = {X 126.3822, Y 92.8094, Z -6.3333, A 0.000, B 0.000, C 0.000 }
gfCNCPoint4[29882] = {X 127.2573, Y 92.5955, Z -6.3333, A 0.000, B 0.000, C 0.000 }
gfCNCPoint4[29883] = {X 128.5206, Y 91.4092, Z -6.3333, A 0.000, B 0.000, C 0.000 }
gfCNCPoint4[29884] = {X 129.7160, Y 90.1544, Z -6.3333, A 0.000, B 0.000, C 0.000 }
gfCNCPoint4[29885] = {X 140.9166, Y 77.8546, Z -6.3333, A 0.000, B 0.000, C 0.000 }
gfCNCPoint4[29886] = {X 137.9000, Y 75.1076, Z -6.3333, A 0.000, B 0.000, C 0.000 }
gfCNCPoint4[29887] = {X 137.9000, Y 75.1076, Z -3.3333, A 0.000, B 0.000, C 0.000 }
gfCNCPoint4[29888] = {X 137.9000, Y 75.1076, Z 11.0000, A 0.000, B 0.000, C 0.000 }
gfCNCPoint4[29889] = {X 165.2864, Y 38.5771, Z 11.0000, A 0.000, B 0.000, C 0.000 }
gfCNCPoint4[29890] = {X 165.2864, Y 38.5771, Z -3.3333, A 0.000, B 0.000, C 0.000 }
gfCNCPoint4[29891] = {X 165.2864, Y 38.5771, Z -6.3333, A 0.000, B 0.000, C 0.000 }
gfCNCPoint4[29892] = {X 169.3156, Y 37.9356, Z -6.3333, A 0.000, B 0.000, C 0.000 }
gfCNCPoint4[29893] = {X 169.2601, Y 37.5869, Z -6.3333, A 0.000, B 0.000, C 0.000 }
gfCNCPoint4[29894] = {X 169.1020, Y 35.9824, Z -6.3333, A 0.000, B 0.000, C 0.000 }
gfCNCPoint4[29895] = {X 169.1190, Y 34.3701, Z -6.3333, A 0.000, B 0.000, C 0.000 }
gfCNCPoint4[29896] = {X 169.3112, Y 32.7692, Z -6.3333, A 0.000, B 0.000, C 0.000 }
gfCNCPoint4[29897] = {X 169.6761, Y 31.1986, Z -6.3333, A 0.000, B 0.000, C 0.000 }
gfCNCPoint4[29898] = {X 170.2094, Y 29.6770, Z -6.3333, A 0.000, B 0.000, C 0.000 }
gfCNCPoint4[29899] = {X 170.8481, Y 28.3701, Z -6.3333, A 0.000, B 0.000, C 0.000 }
gfCNCPoint4[29900] = {X 171.6558, Y 27.1602, Z -6.3333, A 0.000, B 0.000, C 0.000 }
gfCNCPoint4[29901] = {X 172.6181, Y 26.0692, Z -6.3333, A 0.000, B 0.000, C 0.000 }
gfCNCPoint4[29902] = {X 173.7175, Y 25.1167, Z -6.3333, A 0.000, B 0.000, C 0.000 }
gfCNCPoint4[29903] = {X 174.9345, Y 24.3197, Z -6.3333, A 0.000, B 0.000, C 0.000 }
gfCNCPoint4[29904] = {X 174.1520, Y 23.9321, Z -6.3333, A 0.000, B 0.000, C 0.000 }
gfCNCPoint4[29905] = {X 173.4635, Y 23.3950, Z -6.3333, A 0.000, B 0.000, C 0.000 }
gfCNCPoint4[29906] = {X 172.8970, Y 22.7304, Z -6.3333, A 0.000, B 0.000, C 0.000 }
gfCNCPoint4[29907] = {X 172.4758, Y 21.9655, Z -6.3333, A 0.000, B 0.000, C 0.000 }
gfCNCPoint4[29908] = {X 169.8405, Y 15.5121, Z -6.3333, A 0.000, B 0.000, C 0.000 }
gfCNCPoint4[29909] = {X 169.5912, Y 14.6607, Z -6.3333, A 0.000, B 0.000, C 0.000 }
gfCNCPoint4[29910] = {X 169.5212, Y 13.7764, Z -6.3333, A 0.000, B 0.000, C 0.000 }
gfCNCPoint4[29911] = {X 169.6332, Y 12.8964, Z -6.3333, A 0.000, B 0.000, C 0.000 }
gfCNCPoint4[29912] = {X 169.9226, Y 12.0578, Z -6.3333, A 0.000, B 0.000, C 0.000 }
gfCNCPoint4[29913] = {X 170.3773, Y 11.2960, Z -6.3333, A 0.000, B 0.000, C 0.000 }
gfCNCPoint4[29914] = {X 170.9779, Y 10.6432, Z -6.3333, A 0.000, B 0.000, C 0.000 }
gfCNCPoint4[29915] = {X 171.6992, Y 10.1268, Z -6.3333, A 0.000, B 0.000, C 0.000 }
gfCNCPoint4[29916] = {X 172.3295, Y 9.7674, Z -6.3333, A 0.000, B 0.000, C 0.000 }
gfCNCPoint4[29917] = {X 173.1920, Y 9.4018, Z -6.3333, A 0.000, B 0.000, C 0.000 }
gfCNCPoint4[29918] = {X 174.1130, Y 9.2306, Z -6.3333, A 0.000, B 0.000, C 0.000 }
gfCNCPoint4[29919] = {X 175.0493, Y 9.2621, Z -6.3333, A 0.000, B 0.000, C 0.000 }
gfCNCPoint4[29920] = {X 175.9567, Y 9.4946, Z -6.3333, A 0.000, B 0.000, C 0.000 }
gfCNCPoint4[29921] = {X 177.1484, Y 9.0353, Z -6.3333, A 0.000, B 0.000, C 0.000 }
gfCNCPoint4[29922] = {X 179.3258, Y 8.2346, Z -6.3333, A 0.000, B 0.000, C 0.000 }
gfCNCPoint4[29923] = {X 181.5719, Y 7.6540, Z -6.3333, A 0.000, B 0.000, C 0.000 }
gfCNCPoint4[29924] = {X 183.8646, Y 7.2995, Z -6.3333, A 0.000, B 0.000, C 0.000 }
gfCNCPoint4[29925] = {X 186.1812, Y 7.1743, Z -6.3333, A 0.000, B 0.000, C 0.000 }
gfCNCPoint4[29926] = {X 188.4988, Y 7.2799, Z -6.3333, A 0.000, B 0.000, C 0.000 }
gfCNCPoint4[29927] = {X 190.7944, Y 7.6152, Z -6.3333, A 0.000, B 0.000, C 0.000 }
gfCNCPoint4[29928] = {X 192.3686, Y 8.0041, Z -6.3333, A 0.000, B 0.000, C 0.000 }
gfCNCPoint4[29929] = {X 193.8990, Y 8.5404, Z -6.3333, A 0.000, B 0.000, C 0.000 }
gfCNCPoint4[29930] = {X 195.3717, Y 9.2193, Z -6.3333, A 0.000, B 0.000, C 0.000 }
gfCNCPoint4[29931] = {X 196.7734, Y 10.0347, Z -6.3333, A 0.000, B 0.000, C 0.000 }
gfCNCPoint4[29932] = {X 198.0915, Y 10.9792, Z -6.3333, A 0.000, B 0.000, C 0.000 }
gfCNCPoint4[29933] = {X 199.1514, Y 11.9221, Z -6.3333, A 0.000, B 0.000, C 0.000 }
gfCNCPoint4[29934] = {X 200.1023, Y 12.9747, Z -6.3333, A 0.000, B 0.000, C 0.000 }
gfCNCPoint4[29935] = {X 200.9332, Y 14.1244, Z -6.3333, A 0.000, B 0.000, C 0.000 }
gfCNCPoint4[29936] = {X 201.6341, Y 15.3577, Z -6.3333, A 0.000, B 0.000, C 0.000 }
gfCNCPoint4[29937] = {X 202.1967, Y 16.6600, Z -6.3333, A 0.000, B 0.000, C 0.000 }
gfCNCPoint4[29938] = {X 202.6709, Y 18.3163, Z -6.3333, A 0.000, B 0.000, C 0.000 }
gfCNCPoint4[29939] = {X 202.9524, Y 20.0160, Z -6.3333, A 0.000, B 0.000, C 0.000 }
gfCNCPoint4[29940] = {X 203.0374, Y 21.7368, Z -6.3333, A 0.000, B 0.000, C 0.000 }
gfCNCPoint4[29941] = {X 202.9248, Y 23.4560, Z -6.3333, A 0.000, B 0.000, C 0.000 }
gfCNCPoint4[29942] = {X 202.6161, Y 25.1510, Z -6.3333, A 0.000, B 0.000, C 0.000 }
gfCNCPoint4[29943] = {X 202.1742, Y 26.5971, Z -6.3333, A 0.000, B 0.000, C 0.000 }
gfCNCPoint4[29944] = {X 201.5494, Y 27.9742, Z -6.3333, A 0.000, B 0.000, C 0.000 }
gfCNCPoint4[29945] = {X 200.7522, Y 29.2591, Z -6.3333, A 0.000, B 0.000, C 0.000 }
gfCNCPoint4[29946] = {X 199.7958, Y 30.4304, Z -6.3333, A 0.000, B 0.000, C 0.000 }
gfCNCPoint4[29947] = {X 198.6963, Y 31.4686, Z -6.3333, A 0.000, B 0.000, C 0.000 }
gfCNCPoint4[29948] = {X 199.4975, Y 31.8098, Z -6.3333, A 0.000, B 0.000, C 0.000 }
gfCNCPoint4[29949] = {X 200.2139, Y 32.3048, Z -6.3333, A 0.000, B 0.000, C 0.000 }
gfCNCPoint4[29950] = {X 200.8165, Y 32.9335, Z -6.3333, A 0.000, B 0.000, C 0.000 }
gfCNCPoint4[29951] = {X 201.2808, Y 33.6702, Z -6.3333, A 0.000, B 0.000, C 0.000 }
gfCNCPoint4[29952] = {X 204.3222, Y 39.9530, Z -6.3333, A 0.000, B 0.000, C 0.000 }
gfCNCPoint4[29953] = {X 204.6427, Y 40.8622, Z -6.3333, A 0.000, B 0.000, C 0.000 }
gfCNCPoint4[29954] = {X 204.7537, Y 41.8197, Z -6.3333, A 0.000, B 0.000, C 0.000 }
gfCNCPoint4[29955] = {X 204.6496, Y 42.7781, Z -6.3333, A 0.000, B 0.000, C 0.000 }
gfCNCPoint4[29956] = {X 204.3355, Y 43.6895, Z -6.3333, A 0.000, B 0.000, C 0.000 }
gfCNCPoint4[29957] = {X 203.8272, Y 44.5085, Z -6.3333, A 0.000, B 0.000, C 0.000 }
gfCNCPoint4[29958] = {X 203.1499, Y 45.1945, Z -6.3333, A 0.000, B 0.000, C 0.000 }
gfCNCPoint4[29959] = {X 202.6138, Y 45.6279, Z -6.3333, A 0.000, B 0.000, C 0.000 }
gfCNCPoint4[29960] = {X 201.9094, Y 46.0920, Z -6.3333, A 0.000, B 0.000, C 0.000 }
gfCNCPoint4[29961] = {X 201.1283, Y 46.4108, Z -6.3333, A 0.000, B 0.000, C 0.000 }
gfCNCPoint4[29962] = {X 200.3003, Y 46.5721, Z -6.3333, A 0.000, B 0.000, C 0.000 }
gfCNCPoint4[29963] = {X 199.4568, Y 46.5697, Z -6.3333, A 0.000, B 0.000, C 0.000 }
gfCNCPoint4[29964] = {X 198.6297, Y 46.4039, Z -6.3333, A 0.000, B 0.000, C 0.000 }
gfCNCPoint4[29965] = {X 196.5191, Y 47.5047, Z -6.3333, A 0.000, B 0.000, C 0.000 }
gfCNCPoint4[29966] = {X 194.3239, Y 48.4251, Z -6.3333, A 0.000, B 0.000, C 0.000 }
gfCNCPoint4[29967] = {X 192.0594, Y 49.1585, Z -6.3333, A 0.000, B 0.000, C 0.000 }
gfCNCPoint4[29968] = {X 189.8462, Y 49.6711, Z -6.3333, A 0.000, B 0.000, C 0.000 }
gfCNCPoint4[29969] = {X 187.5926, Y 49.9569, Z -6.3333, A 0.000, B 0.000, C 0.000 }
gfCNCPoint4[29970] = {X 185.3216, Y 50.0132, Z -6.3333, A 0.000, B 0.000, C 0.000 }
gfCNCPoint4[29971] = {X 183.0565, Y 49.8392, Z -6.3333, A 0.000, B 0.000, C 0.000 }
gfCNCPoint4[29972] = {X 180.8208, Y 49.4368, Z -6.3333, A 0.000, B 0.000, C 0.000 }
gfCNCPoint4[29973] = {X 178.9807, Y 48.9035, Z -6.3333, A 0.000, B 0.000, C 0.000 }
gfCNCPoint4[29974] = {X 177.2144, Y 48.1615, Z -6.3333, A 0.000, B 0.000, C 0.000 }
gfCNCPoint4[29975] = {X 175.5454, Y 47.2210, Z -6.3333, A 0.000, B 0.000, C 0.000 }
gfCNCPoint4[29976] = {X 173.9959, Y 46.0942, Z -6.3333, A 0.000, B 0.000, C 0.000 }
